C03594=1032.274,-117.414,-80.642,167.484,40.656,157.552
C03595=1032.267,-117.664,-80.633,167.481,40.657,157.552
C03596=1032.262,-117.914,-80.624,167.478,40.658,157.552
C03597=1032.256,-118.163,-80.615,167.476,40.660,157.553
C03598=1032.250,-118.414,-80.606,167.473,40.662,157.553
C03599=1032.245,-118.663,-80.597,167.470,40.663,157.553
C03600=1032.238,-118.913,-80.589,167.467,40.665,157.553
C03601=1032.232,-119.163,-80.579,167.465,40.667,157.553
C03602=1032.226,-119.412,-80.571,167.461,40.668,157.553
C03603=1032.220,-119.662,-80.561,167.458,40.669,157.553
C03604=1032.215,-119.912,-80.553,167.455,40.671,157.553
C03605=1032.208,-120.162,-80.544,167.452,40.673,157.554
C03606=1032.203,-120.411,-80.535,167.450,40.674,157.554
C03607=1032.197,-120.662,-80.526,167.447,40.676,157.554
C03608=1032.191,-120.911,-80.517,167.444,40.678,157.554
C03609=1032.186,-121.161,-80.508,167.441,40.679,157.554
C03610=1032.179,-121.411,-80.499,167.439,40.681,157.554
C03611=1032.173,-121.660,-80.491,167.436,40.682,157.554
C03612=1032.168,-121.911,-80.482,167.433,40.684,157.555
C03613=1032.162,-122.160,-80.473,167.430,40.685,157.555
C03614=1032.155,-122.410,-80.464,167.428,40.687,157.555
C03615=1032.150,-122.660,-80.456,167.425,40.689,157.555
C03616=1032.144,-122.909,-80.446,167.422,40.690,157.555
C03617=1032.139,-123.159,-80.438,167.419,40.692,157.555
C03618=1032.132,-123.409,-80.430,167.417,40.694,157.555
C03619=1032.126,-123.658,-80.420,167.414,40.695,157.556
C03620=1032.121,-123.909,-80.412,167.410,40.697,157.556
C03621=1032.115,-124.158,-80.403,167.407,40.699,157.556
C03622=1032.109,-124.407,-80.394,167.405,40.701,157.556
C03623=1032.103,-124.658,-80.386,167.402,40.702,157.556
C03624=1032.098,-124.907,-80.377,167.399,40.704,157.556
C03625=1032.091,-125.158,-80.369,167.396,40.706,157.556
C03626=1032.086,-125.407,-80.360,167.394,40.707,157.557
C03627=1032.079,-125.657,-80.351,167.391,40.709,157.557
C03628=1032.074,-125.906,-80.343,167.388,40.711,157.557
C03629=1032.068,-126.157,-80.334,167.385,40.712,157.557
C03630=1032.062,-126.406,-80.326,167.383,40.714,157.557
C03631=1032.056,-126.656,-80.317,167.380,40.716,157.557
C03632=1032.051,-126.906,-80.308,167.376,40.717,157.558
C03633=1032.045,-127.155,-80.300,167.373,40.719,157.558
C03634=1032.039,-127.406,-80.291,167.371,40.721,157.558
C03635=1032.033,-127.655,-80.283,167.368,40.722,157.558
C03636=1032.027,-127.904,-80.274,167.365,40.724,157.558
C03637=1032.022,-128.154,-80.266,167.362,40.725,157.558
C03638=1032.017,-128.403,-80.256,167.360,40.726,157.558
C03639=1032.014,-128.653,-80.245,167.357,40.726,157.558
C03640=1032.010,-128.903,-80.235,167.355,40.727,157.558
C03641=1032.008,-129.153,-80.223,167.353,40.725,157.558
C03642=1032.006,-129.403,-80.211,167.351,40.724,157.557
C03643=1032.004,-129.653,-80.199,167.348,40.723,157.557
C03644=1032.004,-129.903,-80.185,167.346,40.721,157.557
C03645=1032.004,-130.152,-80.171,167.344,40.719,157.556
C03646=1032.005,-130.402,-80.157,167.343,40.715,157.556
C03647=1032.006,-130.653,-80.142,167.341,40.712,157.555
C03648=1032.008,-130.902,-80.127,167.339,40.709,157.554
C03649=1032.011,-131.152,-80.111,167.337,40.704,157.553
C03650=1032.014,-131.402,-80.094,167.336,40.699,157.553
C03651=1032.018,-131.653,-80.077,167.335,40.694,157.552
C03652=1032.023,-131.902,-80.059,167.334,40.688,157.551
C03653=1032.029,-132.152,-80.041,167.332,40.682,157.550
C03654=1031.703,-132.177,-80.335,167.284,40.914,157.586
C03655=1031.699,-131.927,-80.354,167.284,40.920,157.587
C03656=1031.694,-131.678,-80.372,167.285,40.927,157.588
C03657=1031.690,-131.428,-80.389,167.288,40.932,157.589
C03658=1031.686,-131.177,-80.406,167.289,40.937,157.590
C03659=1031.683,-130.928,-80.422,167.291,40.941,157.591
C03660=1031.681,-130.677,-80.437,167.291,40.945,157.591
C03661=1031.680,-130.428,-80.452,167.293,40.948,157.592
C03662=1031.679,-130.177,-80.467,167.295,40.951,157.593
C03663=1031.679,-129.927,-80.480,167.298,40.953,157.593
C03664=1031.680,-129.678,-80.494,167.299,40.955,157.594
C03665=1031.681,-129.428,-80.506,167.301,40.957,157.594
C03666=1031.683,-129.178,-80.518,167.304,40.958,157.594
C03667=1031.685,-128.928,-80.529,167.306,40.959,157.594
C03668=1031.689,-128.678,-80.540,167.309,40.959,157.595
C03669=1031.693,-128.428,-80.551,167.311,40.959,157.595
C03670=1031.696,-128.179,-80.561,167.314,40.958,157.595
C03671=1031.702,-127.929,-80.570,167.317,40.956,157.595
C03672=1031.708,-127.679,-80.578,167.320,40.954,157.594
C03673=1031.714,-127.430,-80.587,167.322,40.953,157.594
C03674=1031.719,-127.181,-80.595,167.325,40.951,157.594
C03675=1031.726,-126.931,-80.604,167.328,40.949,157.594
C03676=1031.731,-126.681,-80.612,167.331,40.948,157.594
C03677=1031.736,-126.431,-80.621,167.333,40.946,157.594
C03678=1031.743,-126.182,-80.629,167.336,40.944,157.594
C03679=1031.748,-125.932,-80.638,167.339,40.942,157.593
C03680=1031.755,-125.682,-80.646,167.343,40.941,157.593
C03681=1031.760,-125.432,-80.655,167.345,40.939,157.593
C03682=1031.766,-125.182,-80.664,167.348,40.937,157.593
C03683=1031.772,-124.933,-80.672,167.351,40.936,157.593
C03684=1031.778,-124.683,-80.681,167.353,40.934,157.593
C03685=1031.784,-124.433,-80.690,167.356,40.932,157.593
C03686=1031.790,-124.183,-80.697,167.359,40.931,157.592
C03687=1031.796,-123.934,-80.707,167.362,40.929,157.592
C03688=1031.801,-123.684,-80.715,167.364,40.927,157.592
C03689=1031.807,-123.434,-80.724,167.367,40.925,157.592
C03690=1031.813,-123.184,-80.732,167.371,40.924,157.592
C03691=1031.819,-122.934,-80.742,167.374,40.922,157.592
C03692=1031.824,-122.685,-80.750,167.376,40.920,157.592
C03693=1031.831,-122.434,-80.759,167.379,40.919,157.591
C03694=1031.837,-122.185,-80.768,167.382,40.917,157.591
C03695=1031.842,-121.935,-80.777,167.385,40.915,157.591
C03696=1031.848,-121.686,-80.786,167.387,40.913,157.591
C03697=1031.854,-121.435,-80.795,167.390,40.912,157.591
C03698=1031.860,-121.186,-80.803,167.393,40.910,157.591
C03699=1031.866,-120.936,-80.812,167.396,40.908,157.591
C03700=1031.871,-120.687,-80.821,167.398,40.907,157.590
C03701=1031.877,-120.436,-80.829,167.401,40.905,157.590
C03702=1031.883,-120.187,-80.838,167.405,40.903,157.590
C03703=1031.888,-119.973,-80.846,167.407,40.902,157.590
C03704=1031.893,-119.760,-80.854,167.409,40.901,157.590
C03705=1031.898,-119.546,-80.861,167.411,40.899,157.590
C03706=1031.903,-119.332,-80.869,167.414,40.898,157.590
C03707=1031.908,-119.118,-80.876,167.417,40.896,157.590
C03708=1031.914,-118.904,-80.884,167.419,40.895,157.589
C03709=1031.918,-118.690,-80.892,167.421,40.894,157.589
C03710=1031.924,-118.477,-80.899,167.424,40.892,157.589
C03711=1031.929,-118.226,-80.908,167.427,40.890,157.589
C03712=1031.936,-117.977,-80.918,167.430,40.889,157.589
C03713=1031.942,-117.727,-80.926,167.432,40.887,157.589
C03714=1031.948,-117.477,-80.935,167.435,40.885,157.589
C03715=1031.956,-117.119,-80.949,167.439,40.884,157.589
C03716=1031.965,-116.761,-80.961,167.443,40.881,157.588
C03717=1031.973,-116.403,-80.974,167.447,40.878,157.588
C03718=1031.981,-116.044,-80.987,167.452,40.877,157.588
C03719=1031.987,-115.794,-80.996,167.455,40.875,157.588
C03720=1031.994,-115.544,-81.005,167.457,40.873,157.588
C03721=1031.999,-115.295,-81.014,167.460,40.872,157.588
C03722=1032.005,-115.045,-81.023,167.463,40.870,157.587
C03723=1032.011,-114.795,-81.033,167.466,40.868,157.587
C03724=1032.016,-114.545,-81.041,167.468,40.867,157.587
C03725=1032.023,-114.295,-81.051,167.471,40.865,157.587
C03726=1032.029,-114.045,-81.060,167.474,40.864,157.587
C03727=1032.034,-113.796,-81.069,167.477,40.862,157.587
C03728=1032.040,-113.546,-81.078,167.479,40.860,157.587
C03729=1032.046,-113.296,-81.087,167.482,40.859,157.587
C03730=1032.052,-113.047,-81.096,167.485,40.858,157.586
C03731=1032.058,-112.797,-81.106,167.488,40.856,157.586
C03732=1032.064,-112.547,-81.116,167.491,40.854,157.586
C03733=1032.069,-112.297,-81.124,167.493,40.853,157.586
C03734=1032.075,-112.047,-81.134,167.496,40.852,157.586
C03735=1032.082,-111.798,-81.143,167.499,40.850,157.586
C03736=1032.087,-111.549,-81.152,167.502,40.848,157.586
C03737=1032.093,-111.298,-81.161,167.504,40.847,157.586
C03738=1032.099,-111.048,-81.171,167.508,40.846,157.586
C03739=1032.105,-110.799,-81.180,167.511,40.844,157.585
C03740=1032.111,-110.549,-81.190,167.514,40.842,157.585
C03741=1032.117,-110.299,-81.198,167.516,40.840,157.585
C03742=1032.123,-110.049,-81.208,167.519,40.839,157.585
C03743=1032.129,-109.799,-81.218,167.522,40.838,157.585
C03744=1032.135,-109.550,-81.227,167.525,40.836,157.585
C03745=1032.141,-109.301,-81.236,167.528,40.834,157.585
C03746=1032.147,-109.051,-81.246,167.530,40.833,157.585
C03747=1032.153,-108.800,-81.255,167.533,40.832,157.584
C03748=1032.159,-108.551,-81.264,167.536,40.830,157.584
C03749=1032.165,-108.301,-81.274,167.539,40.828,157.584
C03750=1032.171,-108.052,-81.283,167.542,40.827,157.584
C03751=1032.177,-107.802,-81.293,167.544,40.826,157.584
C03752=1032.183,-107.552,-81.302,167.547,40.824,157.584
C03753=1032.189,-107.302,-81.312,167.550,40.822,157.584
C03754=1032.195,-107.053,-81.321,167.553,40.821,157.584
C03755=1032.200,-106.803,-81.331,167.555,40.820,157.583
C03756=1032.206,-106.553,-81.340,167.558,40.818,157.583
C03757=1032.212,-106.303,-81.350,167.561,40.817,157.583
C03758=1032.219,-106.053,-81.359,167.564,40.815,157.583
C03759=1032.224,-105.804,-81.368,167.567,40.814,157.583
C03760=1032.230,-105.554,-81.378,167.569,40.813,157.583
C03761=1032.236,-105.304,-81.388,167.572,40.811,157.583
C03762=1032.242,-105.054,-81.398,167.575,40.810,157.583
C03763=1032.248,-104.804,-81.407,167.578,40.808,157.583
C03764=1032.254,-104.555,-81.417,167.581,40.807,157.582
C03765=1032.260,-104.306,-81.426,167.583,40.806,157.582
C03766=1032.265,-104.055,-81.436,167.586,40.804,157.582
C03767=1032.272,-103.806,-81.446,167.589,40.803,157.582
C03768=1032.278,-103.556,-81.456,167.592,40.801,157.582
C03769=1032.284,-103.307,-81.466,167.595,40.800,157.582
C03770=1032.290,-103.057,-81.475,167.597,40.799,157.582
C03771=1032.296,-102.807,-81.485,167.600,40.797,157.582
C03772=1032.302,-102.557,-81.495,167.603,40.796,157.582
C03773=1032.308,-102.307,-81.504,167.606,40.794,157.582
C03774=1032.314,-102.058,-81.514,167.609,40.793,157.581
C03775=1032.319,-101.808,-81.524,167.611,40.792,157.581
C03776=1032.325,-101.558,-81.533,167.614,40.790,157.581
C03777=1032.332,-101.309,-81.544,167.617,40.789,157.581
C03778=1032.338,-101.059,-81.553,167.620,40.787,157.581
C03779=1032.344,-100.772,-81.565,167.624,40.785,157.581
C03780=1032.351,-100.485,-81.576,167.626,40.784,157.581
C03781=1032.358,-100.198,-81.587,167.629,40.783,157.581
C03782=1032.365,-99.911,-81.598,167.633,40.781,157.581
C03783=1032.371,-99.661,-81.608,167.636,40.779,157.580
C03784=1032.377,-99.412,-81.618,167.639,40.778,157.580
C03785=1032.383,-99.162,-81.628,167.641,40.777,157.580
C03786=1032.389,-98.912,-81.638,167.644,40.775,157.580
C03787=1032.395,-98.662,-81.648,167.647,40.774,157.580
C03788=1032.401,-98.413,-81.658,167.650,40.772,157.580
C03789=1032.408,-98.163,-81.668,167.653,40.771,157.580
C03790=1032.414,-97.913,-81.677,167.655,40.770,157.580
C03791=1032.419,-97.663,-81.687,167.658,40.768,157.580
C03792=1032.426,-97.414,-81.698,167.661,40.767,157.580
C03793=1032.431,-97.164,-81.708,167.664,40.766,157.580
C03794=1032.437,-96.914,-81.717,167.667,40.764,157.579
C03795=1032.443,-96.665,-81.728,167.670,40.763,157.579
C03796=1032.449,-96.415,-81.738,167.672,40.762,157.579
C03797=1032.455,-96.165,-81.748,167.674,40.761,157.579
C03798=1032.461,-95.916,-81.758,167.677,40.760,157.579
C03799=1032.466,-95.665,-81.768,167.680,40.758,157.579
C03800=1032.473,-95.416,-81.779,167.683,40.757,157.579
C03801=1032.478,-95.166,-81.789,167.686,40.756,157.579
C03802=1032.485,-94.916,-81.798,167.688,40.754,157.579
C03803=1032.490,-94.667,-81.809,167.691,40.753,157.579
C03804=1032.496,-94.417,-81.819,167.694,40.752,157.579
C03805=1032.502,-94.168,-81.830,167.697,40.751,157.579
C03806=1032.508,-93.918,-81.839,167.700,40.750,157.579
C03807=1032.514,-93.668,-81.850,167.702,40.748,157.578
C03808=1032.520,-93.417,-81.861,167.705,40.747,157.578
C03809=1032.527,-93.168,-81.871,167.708,40.746,157.578
C03810=1032.532,-92.918,-81.881,167.711,40.744,157.578
C03811=1032.539,-92.669,-81.891,167.714,40.743,157.578
C03812=1032.544,-92.419,-81.902,167.716,40.742,157.578
C03813=1032.550,-92.170,-81.912,167.718,40.741,157.578
C03814=1032.556,-91.920,-81.922,167.721,40.740,157.578
C03815=1032.562,-91.670,-81.932,167.724,40.738,157.578
C03816=1032.568,-91.420,-81.942,167.727,40.737,157.578
C03817=1032.574,-91.171,-81.953,167.730,40.736,157.578
C03818=1032.580,-90.921,-81.963,167.733,40.734,157.577
C03819=1032.586,-90.671,-81.974,167.736,40.733,157.577
C03820=1032.593,-90.422,-81.984,167.738,40.732,157.577
C03821=1032.598,-90.172,-81.995,167.741,40.731,157.577
C03822=1032.604,-89.922,-82.005,167.744,40.730,157.577
C03823=1032.610,-89.672,-82.015,167.747,40.728,157.577
C03824=1032.616,-89.423,-82.025,167.750,40.727,157.577
C03825=1032.622,-89.174,-82.036,167.752,40.726,157.577
C03826=1032.628,-88.923,-82.047,167.754,40.725,157.577
C03827=1032.635,-88.674,-82.057,167.757,40.724,157.577
C03828=1032.640,-88.423,-82.067,167.760,40.723,157.577
C03829=1032.647,-88.174,-82.077,167.763,40.721,157.577
C03830=1032.652,-87.925,-82.088,167.766,40.720,157.577
C03831=1032.658,-87.674,-82.099,167.768,40.718,157.576
C03832=1032.665,-87.425,-82.109,167.771,40.717,157.576
C03833=1032.671,-87.175,-82.120,167.774,40.716,157.576
C03834=1032.677,-86.926,-82.130,167.777,40.715,157.576
C03835=1032.682,-86.676,-82.140,167.780,40.714,157.576
C03836=1032.689,-86.426,-82.151,167.783,40.713,157.576
C03837=1032.695,-86.177,-82.162,167.786,40.711,157.576
C03838=1032.701,-85.927,-82.172,167.787,40.710,157.576
C03839=1032.707,-85.677,-82.182,167.790,40.709,157.576
C03840=1032.713,-85.427,-82.194,167.793,40.707,157.576
C03841=1032.720,-85.178,-82.204,167.796,40.706,157.576
C03842=1032.725,-84.928,-82.214,167.799,40.705,157.576
C03843=1032.732,-84.643,-82.226,167.802,40.704,157.576
C03844=1032.740,-84.359,-82.239,167.805,40.703,157.575
C03845=1032.746,-84.074,-82.251,167.808,40.701,157.575
C03846=1032.753,-83.789,-82.263,167.811,40.699,157.575
C03847=1032.760,-83.539,-82.274,167.814,40.698,157.575
C03848=1032.766,-83.289,-82.284,167.817,40.697,157.575
C03849=1032.771,-83.040,-82.295,167.819,40.696,157.575
C03850=1032.779,-82.790,-82.305,167.822,40.695,157.575
C03851=1032.784,-82.540,-82.316,167.825,40.694,157.575
C03852=1032.790,-82.291,-82.327,167.828,40.692,157.575
C03853=1032.797,-82.041,-82.338,167.831,40.691,157.575
C03854=1032.803,-81.792,-82.349,167.834,40.690,157.575
C03855=1032.809,-81.542,-82.358,167.837,40.688,157.575
C03856=1032.815,-81.292,-82.369,167.839,40.687,157.574
C03857=1032.821,-81.042,-82.380,167.841,40.687,157.574
C03858=1032.828,-80.793,-82.391,167.844,40.685,157.574
C03859=1032.834,-80.543,-82.402,167.847,40.684,157.574
C03860=1032.840,-80.293,-82.413,167.850,40.683,157.574
C03861=1032.846,-80.044,-82.423,167.853,40.681,157.574
C03862=1032.852,-79.794,-82.434,167.855,40.680,157.574
C03863=1032.858,-79.544,-82.445,167.858,40.679,157.574
C03864=1032.864,-79.295,-82.456,167.861,40.678,157.574
C03865=1032.870,-79.045,-82.467,167.863,40.677,157.574
C03866=1032.876,-78.795,-82.478,167.866,40.676,157.574
C03867=1032.883,-78.545,-82.489,167.869,40.675,157.574
C03868=1032.889,-78.296,-82.500,167.872,40.674,157.574
C03869=1032.895,-78.046,-82.510,167.875,40.673,157.574
C03870=1032.901,-77.796,-82.522,167.877,40.672,157.574
C03871=1032.907,-77.547,-82.533,167.880,40.671,157.574
C03872=1032.912,-77.297,-82.543,167.882,40.670,157.573
C03873=1032.919,-77.047,-82.555,167.885,40.668,157.573
C03874=1032.924,-76.797,-82.566,167.888,40.667,157.573
C03875=1032.932,-76.548,-82.577,167.891,40.666,157.573
C03876=1032.938,-76.299,-82.588,167.894,40.665,157.573
///RCONF 1,0,0,1,0,0,0,0,0,0,0,0,0,0,0,0,0,0,0,0,0,0,0,0
C03877=1032.943,-76.049,-82.599,167.896,40.664,157.573
C03878=1032.950,-75.799,-82.610,167.899,40.663,157.573
C03879=1032.955,-75.550,-82.621,167.901,40.662,157.573
C03880=1032.962,-75.299,-82.632,167.904,40.661,157.573
C03881=1032.968,-75.050,-82.643,167.907,40.660,157.573
C03882=1032.974,-74.800,-82.655,167.910,40.659,157.573
C03883=1032.980,-74.551,-82.666,167.913,40.658,157.573
C03884=1032.986,-74.301,-82.677,167.916,40.657,157.573
C03885=1032.992,-74.051,-82.688,167.917,40.656,157.573
C03886=1032.998,-73.801,-82.699,167.920,40.655,157.573
C03887=1033.004,-73.552,-82.711,167.923,40.654,157.573
C03888=1033.010,-73.303,-82.722,167.926,40.653,157.573
C03889=1033.016,-73.052,-82.733,167.929,40.652,157.573
C03890=1033.022,-72.803,-82.744,167.931,40.651,157.573
C03891=1033.028,-72.553,-82.756,167.934,40.650,157.572
C03892=1033.034,-72.303,-82.767,167.937,40.649,157.572
C03893=1033.040,-72.054,-82.779,167.940,40.648,157.572
C03894=1033.046,-71.804,-82.790,167.941,40.647,157.572
C03895=1033.053,-71.554,-82.801,167.944,40.646,157.572
C03896=1033.058,-71.305,-82.813,167.947,40.645,157.572
C03897=1033.064,-71.055,-82.825,167.950,40.644,157.572
///RCONF 1,0,0,0,0,0,0,0,0,0,0,0,0,0,0,0,0,0,0,0,0,0,0,0
C03898=1033.070,-70.805,-82.836,167.953,40.643,157.572
C03899=1033.077,-70.556,-82.848,167.955,40.642,157.572
C03900=1033.082,-70.306,-82.858,167.958,40.642,157.572
C03901=1033.088,-70.056,-82.871,167.961,40.641,157.572
C03902=1033.094,-69.807,-82.882,167.964,40.640,157.572
C03903=1033.100,-69.557,-82.893,167.966,40.639,157.572
C03904=1033.106,-69.308,-82.905,167.968,40.638,157.572
C03905=1033.113,-69.058,-82.916,167.971,40.637,157.572
C03906=1033.118,-68.808,-82.928,167.974,40.636,157.572
C03907=1033.125,-68.526,-82.941,167.977,40.635,157.572
C03908=1033.132,-68.243,-82.954,167.980,40.634,157.572
C03909=1033.139,-67.961,-82.967,167.983,40.633,157.572
C03910=1033.146,-67.677,-82.980,167.986,40.632,157.572
C03911=1033.151,-67.428,-82.991,167.989,40.631,157.572
C03912=1033.158,-67.178,-83.003,167.992,40.630,157.572
C03913=1033.164,-66.929,-83.014,167.994,40.629,157.572
C03914=1033.170,-66.679,-83.026,167.996,40.629,157.572
C03915=1033.176,-66.429,-83.037,167.999,40.628,157.572
C03916=1033.182,-66.180,-83.050,168.002,40.627,157.572
C03917=1033.189,-65.930,-83.062,168.005,40.626,157.572
C03918=1033.194,-65.681,-83.072,168.007,40.625,157.571
C03919=1033.201,-65.431,-83.084,168.010,40.624,157.571
C03920=1033.206,-65.181,-83.096,168.013,40.623,157.571
C03921=1033.213,-64.932,-83.108,168.016,40.622,157.571
C03922=1033.219,-64.681,-83.119,168.017,40.621,157.571
C03923=1033.225,-64.433,-83.131,168.020,40.620,157.571
C03924=1033.231,-64.183,-83.143,168.023,40.619,157.571
C03925=1033.237,-63.932,-83.154,168.026,40.618,157.571
C03926=1033.243,-63.684,-83.166,168.028,40.617,157.571
C03927=1033.250,-63.433,-83.177,168.031,40.616,157.571
C03928=1033.256,-63.184,-83.189,168.034,40.615,157.571
C03929=1033.262,-62.935,-83.201,168.037,40.615,157.571
C03930=1033.268,-62.684,-83.213,168.040,40.614,157.571
C03931=1033.275,-62.435,-83.225,168.042,40.613,157.571
C03932=1033.281,-62.186,-83.236,168.044,40.612,157.571
C03933=1033.286,-61.935,-83.248,168.047,40.611,157.571
C03934=1033.293,-61.686,-83.260,168.050,40.610,157.571
C03935=1033.299,-61.437,-83.272,168.052,40.609,157.571
C03936=1033.305,-61.187,-83.283,168.055,40.608,157.571
C03937=1033.311,-60.937,-83.295,168.058,40.607,157.571
C03938=1033.318,-60.687,-83.307,168.061,40.606,157.571
C03939=1033.324,-60.438,-83.318,168.063,40.605,157.571
C03940=1033.330,-60.188,-83.331,168.066,40.604,157.571
C03941=1033.336,-59.938,-83.343,168.068,40.603,157.571
C03942=1033.343,-59.689,-83.355,168.071,40.602,157.571
C03943=1033.349,-59.439,-83.366,168.073,40.602,157.570
C03944=1033.354,-59.190,-83.378,168.076,40.601,157.570
C03945=1033.361,-58.940,-83.390,168.079,40.600,157.570
C03946=1033.368,-58.690,-83.402,168.082,40.599,157.571
C03947=1033.373,-58.441,-83.414,168.084,40.598,157.570
C03948=1033.379,-58.191,-83.425,168.087,40.597,157.570
C03949=1033.386,-57.941,-83.437,168.090,40.596,157.570
C03950=1033.393,-57.692,-83.449,168.092,40.596,157.570
C03951=1033.399,-57.442,-83.462,168.094,40.595,157.570
C03952=1033.405,-57.193,-83.474,168.097,40.594,157.570
C03953=1033.411,-56.943,-83.485,168.100,40.593,157.570
C03954=1033.417,-56.693,-83.497,168.102,40.592,157.570
C03955=1033.424,-56.443,-83.509,168.105,40.591,157.570
C03956=1033.430,-56.194,-83.521,168.108,40.590,157.570
C03957=1033.436,-55.945,-83.533,168.111,40.589,157.570
C03958=1033.442,-55.695,-83.545,168.113,40.588,157.570
C03959=1033.449,-55.446,-83.557,168.116,40.587,157.570
C03960=1033.455,-55.195,-83.569,168.118,40.586,157.570
C03961=1033.461,-54.945,-83.581,168.121,40.585,157.570
C03962=1033.468,-54.696,-83.593,168.123,40.585,157.570
C03963=1033.474,-54.446,-83.605,168.126,40.584,157.570
C03964=1033.480,-54.197,-83.617,168.129,40.583,157.570
C03965=1033.486,-53.948,-83.629,168.132,40.582,157.570
C03966=1033.493,-53.698,-83.641,168.134,40.581,157.570
C03967=1033.499,-53.448,-83.654,168.137,40.580,157.570
C03968=1033.505,-53.199,-83.666,168.140,40.579,157.570
C03969=1033.512,-52.949,-83.678,168.142,40.578,157.570
C03970=1033.519,-52.699,-83.690,168.144,40.577,157.570
C03971=1033.525,-52.418,-83.703,168.147,40.576,157.569
C03972=1033.533,-52.137,-83.717,168.150,40.575,157.569
C03973=1033.540,-51.855,-83.731,168.153,40.574,157.569
C03974=1033.547,-51.574,-83.744,168.156,40.573,157.569
C03975=1033.553,-51.324,-83.757,168.159,40.572,157.569
C03976=1033.560,-51.075,-83.769,168.162,40.571,157.569
C03977=1033.566,-50.825,-83.781,168.165,40.570,157.569
C03978=1033.572,-50.575,-83.794,168.167,40.569,157.569
C03979=1033.579,-50.326,-83.806,168.169,40.568,157.569
C03980=1033.585,-50.076,-83.818,168.173,40.568,157.569
C03981=1033.591,-49.826,-83.831,168.174,40.567,157.569
C03982=1033.597,-49.576,-83.843,168.177,40.566,157.569
C03983=1033.603,-49.327,-83.855,168.180,40.566,157.569
C03984=1033.609,-49.078,-83.868,168.182,40.565,157.569
C03985=1033.616,-48.828,-83.880,168.185,40.564,157.569
C03986=1033.621,-48.578,-83.893,168.187,40.563,157.569
C03987=1033.627,-48.329,-83.905,168.190,40.563,157.569
C03988=1033.634,-48.079,-83.917,168.193,40.562,157.569
C03989=1033.640,-47.830,-83.930,168.195,40.561,157.569
C03990=1033.646,-47.580,-83.943,168.198,40.561,157.569
C03991=1033.652,-47.330,-83.955,168.201,40.560,157.569
C03992=1033.659,-47.080,-83.967,168.203,40.559,157.569
C03993=1033.665,-46.831,-83.981,168.206,40.559,157.569
C03994=1033.671,-46.581,-83.993,168.209,40.558,157.569
C03995=1033.677,-46.332,-84.005,168.210,40.557,157.569
C03996=1033.683,-46.082,-84.018,168.213,40.556,157.569
C03997=1033.690,-45.833,-84.031,168.215,40.556,157.569
C03998=1033.696,-45.583,-84.043,168.218,40.555,157.569
C03999=1033.702,-45.333,-84.056,168.221,40.554,157.569
C04000=1033.708,-45.084,-84.069,168.223,40.553,157.569
C04001=1033.714,-44.834,-84.081,168.226,40.552,157.569
C04002=1033.721,-44.584,-84.093,168.229,40.551,157.569
C04003=1033.727,-44.335,-84.107,168.231,40.551,157.569
C04004=1033.733,-44.085,-84.119,168.234,40.550,157.569
C04005=1033.740,-43.836,-84.131,168.236,40.549,157.569
C04006=1033.746,-43.586,-84.144,168.239,40.549,157.569
C04007=1033.752,-43.337,-84.157,168.242,40.548,157.569
C04008=1033.758,-43.087,-84.170,168.244,40.547,157.569
C04009=1033.765,-42.838,-84.182,168.246,40.546,157.569
C04010=1033.771,-42.588,-84.195,168.249,40.546,157.569
C04011=1033.777,-42.339,-84.208,168.251,40.545,157.569
C04012=1033.783,-42.089,-84.221,168.254,40.544,157.569
C04013=1033.790,-41.840,-84.233,168.256,40.544,157.569
C04014=1033.796,-41.590,-84.246,168.259,40.543,157.569
C04015=1033.802,-41.339,-84.259,168.262,40.542,157.569
C04016=1033.808,-41.090,-84.272,168.264,40.542,157.569
C04017=1033.815,-40.840,-84.284,168.267,40.541,157.569
C04018=1033.821,-40.591,-84.297,168.270,40.540,157.569
C04019=1033.827,-40.341,-84.310,168.272,40.539,157.569
C04020=1033.833,-40.092,-84.323,168.275,40.539,157.569
C04021=1033.840,-39.842,-84.335,168.277,40.538,157.569
C04022=1033.846,-39.593,-84.348,168.279,40.537,157.569
C04023=1033.852,-39.343,-84.361,168.283,40.536,157.569
C04024=1033.859,-39.093,-84.374,168.284,40.536,157.569
C04025=1033.865,-38.844,-84.386,168.287,40.535,157.569
C04026=1033.872,-38.594,-84.400,168.289,40.534,157.569
C04027=1033.878,-38.345,-84.412,168.292,40.533,157.569
C04028=1033.884,-38.095,-84.426,168.295,40.533,157.569
C04029=1033.890,-37.846,-84.439,168.297,40.532,157.569
C04030=1033.896,-37.596,-84.451,168.300,40.531,157.569
C04031=1033.903,-37.346,-84.465,168.302,40.531,157.569
C04032=1033.909,-37.097,-84.478,168.305,40.530,157.569
C04033=1033.915,-36.847,-84.491,168.307,40.530,157.569
C04034=1033.921,-36.598,-84.504,168.310,40.529,157.569
C04035=1033.928,-36.316,-84.519,168.313,40.529,157.569
C04036=1033.935,-36.036,-84.534,168.316,40.528,157.569
C04037=1033.942,-35.755,-84.548,168.319,40.527,157.569
C04038=1033.948,-35.474,-84.563,168.321,40.526,157.569
C04039=1033.954,-35.224,-84.576,168.324,40.526,157.569
C04040=1033.961,-34.974,-84.590,168.327,40.525,157.569
C04041=1033.967,-34.724,-84.602,168.328,40.524,157.569
C04042=1033.973,-34.475,-84.616,168.332,40.524,157.569
C04043=1033.979,-34.226,-84.629,168.333,40.523,157.569
C04044=1033.986,-33.977,-84.642,168.336,40.522,157.569
C04045=1033.992,-33.726,-84.655,168.338,40.522,157.569
C04046=1033.998,-33.477,-84.668,168.341,40.521,157.569
C04047=1034.005,-33.228,-84.682,168.343,40.521,157.569
C04048=1034.011,-32.978,-84.695,168.346,40.520,157.569
C04049=1034.017,-32.728,-84.708,168.348,40.520,157.569
C04050=1034.024,-32.478,-84.721,168.351,40.519,157.569
C04051=1034.030,-32.229,-84.734,168.354,40.518,157.569
C04052=1034.036,-31.980,-84.748,168.356,40.517,157.569
C04053=1034.043,-31.730,-84.761,168.359,40.516,157.569
C04054=1034.049,-31.480,-84.774,168.361,40.516,157.569
C04055=1034.055,-31.231,-84.787,168.364,40.515,157.569
C04056=1034.061,-30.982,-84.800,168.366,40.515,157.569
C04057=1034.068,-30.732,-84.814,168.369,40.514,157.569
C04058=1034.074,-30.482,-84.827,168.371,40.514,157.569
C04059=1034.080,-30.233,-84.841,168.374,40.513,157.569
C04060=1034.087,-29.984,-84.854,168.375,40.512,157.569
C04061=1034.093,-29.733,-84.867,168.379,40.512,157.569
C04062=1034.099,-29.484,-84.880,168.380,40.511,157.569
C04063=1034.106,-29.235,-84.893,168.383,40.511,157.569
C04064=1034.112,-28.985,-84.907,168.386,40.510,157.569
C04065=1034.119,-28.735,-84.920,168.388,40.509,157.569
C04066=1034.125,-28.486,-84.933,168.391,40.508,157.569
C04067=1034.131,-28.236,-84.948,168.393,40.508,157.569
C04068=1034.137,-27.987,-84.961,168.396,40.507,157.569
C04069=1034.143,-27.737,-84.974,168.398,40.506,157.569
C04070=1034.150,-27.487,-84.988,168.401,40.506,157.569
C04071=1034.156,-27.238,-85.001,168.403,40.505,157.569
C04072=1034.163,-26.989,-85.014,168.406,40.505,157.569
C04073=1034.169,-26.739,-85.028,168.408,40.504,157.569
C04074=1034.175,-26.489,-85.042,168.411,40.504,157.569
C04075=1034.181,-26.240,-85.055,168.413,40.503,157.569
C04076=1034.188,-25.990,-85.069,168.416,40.503,157.569
C04077=1034.193,-25.741,-85.083,168.418,40.502,157.569
C04078=1034.200,-25.491,-85.096,168.421,40.501,157.569
C04079=1034.206,-25.241,-85.110,168.423,40.501,157.569
C04080=1034.213,-24.992,-85.123,168.426,40.500,157.569
C04081=1034.218,-24.742,-85.137,168.428,40.500,157.569
C04082=1034.225,-24.492,-85.150,168.431,40.499,157.569
C04083=1034.231,-24.243,-85.164,168.433,40.499,157.569
C04084=1034.237,-23.993,-85.178,168.435,40.499,157.569
C04085=1034.243,-23.744,-85.191,168.437,40.498,157.569
C04086=1034.250,-23.495,-85.205,168.440,40.497,157.569
C04087=1034.256,-23.245,-85.219,168.442,40.497,157.569
C04088=1034.262,-22.995,-85.233,168.444,40.496,157.569
C04089=1034.268,-22.746,-85.246,168.447,40.496,157.569
C04090=1034.274,-22.496,-85.260,168.449,40.495,157.569
C04091=1034.281,-22.247,-85.273,168.452,40.495,157.569
C04092=1034.288,-21.997,-85.288,168.454,40.494,157.569
C04093=1034.293,-21.748,-85.302,168.457,40.494,157.569
C04094=1034.300,-21.499,-85.315,168.459,40.493,157.569
C04095=1034.306,-21.249,-85.329,168.462,40.492,157.569
C04096=1034.312,-20.999,-85.342,168.464,40.492,157.569
C04097=1034.319,-20.750,-85.357,168.467,40.491,157.569
C04098=1034.325,-20.500,-85.370,168.469,40.491,157.569
C04099=1034.332,-20.218,-85.385,168.472,40.490,157.569
C04100=1034.339,-19.937,-85.401,168.475,40.490,157.569
C04101=1034.347,-19.654,-85.417,168.477,40.489,157.569
C04102=1034.353,-19.373,-85.432,168.480,40.489,157.569
C04103=1034.360,-19.123,-85.446,168.483,40.488,157.569
C04104=1034.366,-18.874,-85.460,168.485,40.487,157.569
C04105=1034.373,-18.624,-85.474,168.487,40.487,157.569
C04106=1034.378,-18.375,-85.488,168.490,40.486,157.569
C04107=1034.385,-18.125,-85.502,168.492,40.485,157.569
C04108=1034.392,-17.876,-85.516,168.495,40.485,157.569
C04109=1034.398,-17.626,-85.530,168.497,40.485,157.569
C04110=1034.404,-17.377,-85.543,168.500,40.484,157.569
C04111=1034.411,-17.127,-85.557,168.502,40.484,157.569
C04112=1034.417,-16.878,-85.571,168.505,40.483,157.569
C04113=1034.423,-16.628,-85.585,168.507,40.483,157.569
C04114=1034.429,-16.379,-85.600,168.509,40.482,157.569
C04115=1034.436,-16.129,-85.613,168.511,40.481,157.569
C04116=1034.442,-15.880,-85.627,168.513,40.481,157.569
C04117=1034.449,-15.630,-85.641,168.516,40.480,157.569
C04118=1034.455,-15.380,-85.655,168.518,40.479,157.569
C04119=1034.461,-15.131,-85.670,168.521,40.479,157.569
C04120=1034.468,-14.881,-85.683,168.523,40.479,157.569
C04121=1034.474,-14.632,-85.698,168.525,40.479,157.569
C04122=1034.481,-14.382,-85.711,168.528,40.478,157.569
C04123=1034.486,-14.133,-85.726,168.530,40.477,157.569
C04124=1034.492,-13.883,-85.740,168.533,40.477,157.569
C04125=1034.499,-13.634,-85.754,168.535,40.476,157.569
C04126=1034.505,-13.384,-85.768,168.537,40.476,157.569
C04127=1034.511,-13.135,-85.783,168.540,40.476,157.569
C04128=1034.518,-12.885,-85.797,168.542,40.475,157.569
C04129=1034.523,-12.636,-85.811,168.545,40.475,157.570
C04130=1034.530,-12.386,-85.825,168.547,40.474,157.570
C04131=1034.537,-12.136,-85.840,168.549,40.474,157.569
C04132=1034.542,-11.887,-85.854,168.552,40.473,157.570
C04133=1034.549,-11.638,-85.868,168.554,40.473,157.570
C04134=1034.555,-11.389,-85.883,168.557,40.473,157.570
C04135=1034.562,-11.139,-85.896,168.559,40.472,157.570
C04136=1034.568,-10.890,-85.911,168.561,40.472,157.570
C04137=1034.574,-10.639,-85.925,168.564,40.471,157.570
C04138=1034.581,-10.390,-85.939,168.566,40.470,157.570
C04139=1034.587,-10.141,-85.954,168.569,40.470,157.570
C04140=1034.593,-9.891,-85.968,168.571,40.470,157.570
C04141=1034.600,-9.641,-85.983,168.573,40.469,157.570
C04142=1034.605,-9.392,-85.996,168.576,40.469,157.570
C04143=1034.612,-9.142,-86.011,168.578,40.469,157.570
C04144=1034.618,-8.894,-86.025,168.580,40.468,157.570
C04145=1034.624,-8.643,-86.040,168.583,40.467,157.570
C04146=1034.631,-8.394,-86.055,168.585,40.467,157.570
C04147=1034.637,-8.145,-86.069,168.588,40.466,157.570
C04148=1034.643,-7.895,-86.083,168.590,40.466,157.570
C04149=1034.650,-7.645,-86.097,168.592,40.466,157.570
C04150=1034.656,-7.396,-86.112,168.595,40.465,157.570
C04151=1034.662,-7.146,-86.126,168.597,40.465,157.570
C04152=1034.669,-6.897,-86.140,168.599,40.464,157.570
C04153=1034.675,-6.648,-86.155,168.602,40.464,157.570
C04154=1034.681,-6.398,-86.170,168.604,40.463,157.570
C04155=1034.688,-6.148,-86.183,168.607,40.463,157.570
C04156=1034.695,-5.899,-86.198,168.609,40.462,157.570
C04157=1034.700,-5.650,-86.213,168.611,40.462,157.570
C04158=1034.708,-5.400,-86.227,168.614,40.461,157.570
C04159=1034.714,-5.150,-86.242,168.616,40.461,157.570
C04160=1034.719,-4.901,-86.256,168.618,40.461,157.570
C04161=1034.727,-4.652,-86.271,168.620,40.460,157.570
C04162=1034.733,-4.402,-86.285,168.622,40.459,157.570
C04163=1034.740,-4.119,-86.302,168.626,40.459,157.570
C04164=1034.747,-3.835,-86.318,168.628,40.458,157.570
C04165=1034.754,-3.552,-86.335,168.630,40.458,157.570
C04166=1034.762,-3.269,-86.352,168.633,40.458,157.570
C04167=1034.768,-3.019,-86.367,168.635,40.457,157.570
C04168=1034.774,-2.769,-86.381,168.639,40.457,157.571
C04169=1034.780,-2.520,-86.395,168.640,40.456,157.570
C04170=1034.786,-2.270,-86.410,168.642,40.456,157.571
C04171=1034.793,-2.021,-86.425,168.644,40.456,157.571
C04172=1034.798,-1.772,-86.440,168.647,40.456,157.571
C04173=1034.805,-1.522,-86.455,168.650,40.455,157.571
C04174=1034.811,-1.272,-86.470,168.652,40.455,157.571
C04175=1034.817,-1.023,-86.485,168.654,40.454,157.571
C04176=1034.823,-0.774,-86.499,168.656,40.454,157.571
C04177=1034.830,-0.524,-86.514,168.658,40.454,157.571
C04178=1034.836,-0.274,-86.529,168.662,40.453,157.571
C04179=1034.842,-0.025,-86.544,168.664,40.453,157.571
C04180=1034.848,0.224,-86.559,168.666,40.453,157.571
C04181=1034.855,0.474,-86.574,168.667,40.452,157.571
C04182=1034.861,0.724,-86.589,168.670,40.452,157.571
C04183=1034.867,0.973,-86.603,168.672,40.452,157.571
C04184=1034.873,1.222,-86.618,168.675,40.451,157.571
C04185=1034.880,1.472,-86.633,168.678,40.451,157.571
C04186=1034.886,1.722,-86.648,168.680,40.451,157.571
C04187=1034.892,1.971,-86.663,168.681,40.450,157.571
C04188=1034.899,2.220,-86.679,168.684,40.450,157.571
C04189=1034.905,2.469,-86.693,168.687,40.450,157.571
C04190=1034.911,2.719,-86.708,168.689,40.449,157.571
C04191=1034.918,2.968,-86.723,168.691,40.449,157.571
C04192=1034.924,3.218,-86.738,168.693,40.448,157.571
C04193=1034.930,3.468,-86.753,168.695,40.448,157.571
C04194=1034.936,3.717,-86.768,168.697,40.448,157.571
C04195=1034.942,3.966,-86.782,168.701,40.447,157.572
C04196=1034.948,4.216,-86.798,168.703,40.447,157.572
C04197=1034.955,4.465,-86.814,168.704,40.446,157.572
C04198=1034.961,4.715,-86.829,168.706,40.446,157.572
C04199=1034.968,4.965,-86.844,168.709,40.446,157.572
C04200=1034.973,5.214,-86.858,168.712,40.446,157.572
C04201=1034.980,5.463,-86.873,168.714,40.446,157.572
C04202=1034.986,5.713,-86.888,168.716,40.445,157.572
C04203=1034.993,5.962,-86.904,168.718,40.444,157.572
C04204=1034.999,6.212,-86.919,168.720,40.444,157.572
C04205=1035.006,6.461,-86.934,168.723,40.444,157.572
C04206=1035.012,6.711,-86.949,168.726,40.444,157.572
C04207=1035.018,6.961,-86.963,168.727,40.443,157.572
C04208=1035.025,7.210,-86.979,168.729,40.443,157.572
C04209=1035.031,7.459,-86.994,168.732,40.442,157.572
C04210=1035.037,7.708,-87.009,168.734,40.442,157.572
C04211=1035.044,7.958,-87.024,168.736,40.441,157.572
C04212=1035.050,8.207,-87.039,168.738,40.441,157.572
C04213=1035.057,8.457,-87.054,168.741,40.441,157.572
C04214=1035.063,8.706,-87.069,168.743,40.440,157.572
C04215=1035.069,8.956,-87.084,168.745,40.440,157.572
C04216=1035.076,9.205,-87.100,168.748,40.439,157.572
C04217=1035.082,9.455,-87.115,168.750,40.439,157.572
C04218=1035.088,9.705,-87.130,168.752,40.439,157.572
C04219=1035.094,9.954,-87.145,168.754,40.439,157.572
C04220=1035.101,10.203,-87.161,168.757,40.438,157.572
C04221=1035.108,10.453,-87.176,168.759,40.438,157.572
C04222=1035.114,10.703,-87.191,168.761,40.437,157.572
C04223=1035.121,10.952,-87.206,168.764,40.437,157.573
C04224=1035.127,11.201,-87.221,168.766,40.436,157.572
C04225=1035.133,11.451,-87.236,168.768,40.436,157.572
C04226=1035.140,11.700,-87.252,168.770,40.436,157.573
C04227=1035.147,11.985,-87.269,168.773,40.435,157.573
C04228=1035.154,12.270,-87.286,168.776,40.434,157.573
C04229=1035.162,12.556,-87.304,168.778,40.434,157.573
C04230=1035.169,12.841,-87.322,168.781,40.434,157.573
C04231=1035.176,13.090,-87.337,168.783,40.434,157.573
C04232=1035.182,13.339,-87.352,168.785,40.433,157.573
C04233=1035.189,13.589,-87.367,168.788,40.433,157.573
C04234=1035.194,13.839,-87.383,168.790,40.432,157.573
C04235=1035.201,14.088,-87.398,168.792,40.432,157.573
C04236=1035.208,14.338,-87.413,168.794,40.431,157.573
C04237=1035.213,14.587,-87.430,168.797,40.431,157.573
C04238=1035.220,14.837,-87.445,168.799,40.431,157.573
C04239=1035.227,15.086,-87.460,168.801,40.431,157.573
C04240=1035.232,15.336,-87.476,168.803,40.430,157.573
C04241=1035.239,15.585,-87.491,168.806,40.430,157.573
C04242=1035.245,15.835,-87.506,168.808,40.430,157.573
C04243=1035.251,16.084,-87.523,168.810,40.430,157.573
C04244=1035.258,16.333,-87.538,168.812,40.430,157.573
C04245=1035.264,16.583,-87.553,168.814,40.429,157.573
C04246=1035.270,16.832,-87.569,168.817,40.428,157.573
C04247=1035.277,17.082,-87.584,168.819,40.428,157.573
C04248=1035.283,17.331,-87.600,168.821,40.428,157.573
C04249=1035.289,17.581,-87.616,168.823,40.428,157.573
C04250=1035.296,17.830,-87.632,168.826,40.427,157.574
C04251=1035.303,18.079,-87.647,168.828,40.427,157.574
C04252=1035.309,18.329,-87.663,168.830,40.427,157.574
C04253=1035.315,18.578,-87.678,168.832,40.426,157.574
C04254=1035.322,18.827,-87.694,168.834,40.426,157.574
C04255=1035.328,19.077,-87.710,168.837,40.426,157.574
C04256=1035.334,19.326,-87.725,168.839,40.425,157.574
C04257=1035.341,19.576,-87.740,168.841,40.425,157.574
C04258=1035.347,19.825,-87.757,168.843,40.425,157.574
C04259=1035.353,20.074,-87.772,168.845,40.425,157.574
C04260=1035.359,20.324,-87.788,168.849,40.425,157.574
C04261=1035.366,20.573,-87.803,168.851,40.424,157.574
C04262=1035.372,20.823,-87.820,168.852,40.423,157.574
C04263=1035.379,21.073,-87.836,168.854,40.423,157.574
C04264=1035.385,21.323,-87.851,168.856,40.423,157.574
C04265=1035.391,21.572,-87.867,168.859,40.423,157.574
C04266=1035.397,21.821,-87.883,168.862,40.423,157.574
C04267=1035.404,22.070,-87.899,168.864,40.422,157.574
C04268=1035.410,22.319,-87.915,168.866,40.422,157.574
C04269=1035.416,22.569,-87.930,168.868,40.422,157.574
C04270=1035.422,22.818,-87.946,168.871,40.422,157.574
C04271=1035.429,23.067,-87.962,168.873,40.421,157.574
C04272=1035.435,23.317,-87.979,168.875,40.421,157.575
C04273=1035.442,23.567,-87.994,168.877,40.421,157.575
C04274=1035.448,23.816,-88.010,168.879,40.421,157.575
C04275=1035.454,24.065,-88.025,168.882,40.420,157.575
C04276=1035.460,24.315,-88.042,168.884,40.420,157.575
C04277=1035.467,24.564,-88.057,168.886,40.419,157.575
C04278=1035.473,24.813,-88.074,168.888,40.419,157.575
C04279=1035.480,25.064,-88.089,168.890,40.419,157.575
C04280=1035.486,25.313,-88.105,168.893,40.419,157.575
C04281=1035.492,25.562,-88.121,168.895,40.419,157.575
C04282=1035.499,25.811,-88.137,168.897,40.418,157.575
C04283=1035.505,26.061,-88.153,168.899,40.418,157.575
C04284=1035.512,26.310,-88.169,168.901,40.418,157.575
C04285=1035.518,26.560,-88.186,168.904,40.417,157.575
C04286=1035.524,26.809,-88.201,168.906,40.417,157.575
C04287=1035.530,27.058,-88.218,168.908,40.417,157.575
C04288=1035.537,27.308,-88.232,168.910,40.416,157.575
C04289=1035.543,27.558,-88.249,168.912,40.416,157.575
C04290=1035.549,27.807,-88.265,168.914,40.416,157.575
C04291=1035.557,28.093,-88.284,168.917,40.416,157.575
C04292=1035.564,28.380,-88.303,168.919,40.415,157.575
C04293=1035.571,28.666,-88.321,168.922,40.415,157.575
C04294=1035.579,28.953,-88.339,168.924,40.415,157.576
C04295=1035.585,29.202,-88.355,168.927,40.415,157.576
C04296=1035.590,29.451,-88.372,168.929,40.414,157.576
C04297=1035.598,29.701,-88.388,168.931,40.414,157.576
C04298=1035.604,29.951,-88.404,168.933,40.414,157.576
C04299=1035.610,30.200,-88.420,168.935,40.414,157.576
C04300=1035.616,30.449,-88.437,168.937,40.414,157.576
C04301=1035.623,30.699,-88.453,168.939,40.413,157.576
C04302=1035.629,30.948,-88.469,168.942,40.413,157.576
C04303=1035.635,31.197,-88.486,168.944,40.413,157.576
C04304=1035.641,31.446,-88.502,168.946,40.413,157.576
C04305=1035.648,31.696,-88.518,168.948,40.413,157.576
C04306=1035.654,31.945,-88.534,168.950,40.412,157.576
C04307=1035.660,32.195,-88.551,168.952,40.412,157.576
C04308=1035.666,32.444,-88.567,168.955,40.412,157.576
C04309=1035.673,32.694,-88.583,168.957,40.412,157.576
C04310=1035.679,32.943,-88.599,168.959,40.411,157.576
C04311=1035.685,33.193,-88.615,168.961,40.411,157.577
C04312=1035.692,33.441,-88.632,168.963,40.411,157.577
C04313=1035.698,33.691,-88.649,168.965,40.411,157.577
C04314=1035.705,33.940,-88.665,168.967,40.410,157.577
C04315=1035.711,34.190,-88.681,168.970,40.410,157.577
C04316=1035.717,34.440,-88.698,168.972,40.409,157.577
C04317=1035.723,34.689,-88.714,168.974,40.409,157.577
C04318=1035.730,34.938,-88.730,168.976,40.409,157.577
C04319=1035.737,35.188,-88.747,168.978,40.409,157.577
C04320=1035.743,35.437,-88.763,168.980,40.409,157.577
C04321=1035.749,35.686,-88.779,168.982,40.408,157.577
C04322=1035.755,35.936,-88.796,168.985,40.408,157.577
C04323=1035.762,36.185,-88.812,168.988,40.408,157.577
C04324=1035.768,36.434,-88.829,168.990,40.408,157.577
C04325=1035.775,36.684,-88.845,168.992,40.407,157.577
C04326=1035.781,36.934,-88.861,168.994,40.407,157.577
C04327=1035.787,37.182,-88.878,168.996,40.407,157.577
C04328=1035.794,37.432,-88.894,168.999,40.407,157.577
C04329=1035.800,37.681,-88.911,169.001,40.407,157.577
C04330=1035.807,37.930,-88.928,169.003,40.406,157.577
C04331=1035.813,38.180,-88.944,169.005,40.406,157.578
C04332=1035.819,38.429,-88.961,169.007,40.406,157.578
C04333=1035.825,38.678,-88.977,169.009,40.406,157.578
C04334=1035.832,38.928,-88.994,169.011,40.406,157.578
C04335=1035.838,39.178,-89.010,169.013,40.405,157.578
C04336=1035.844,39.426,-89.027,169.015,40.405,157.578
C04337=1035.851,39.676,-89.044,169.018,40.405,157.578
C04338=1035.857,39.926,-89.060,169.020,40.405,157.578
C04339=1035.862,40.175,-89.078,169.022,40.404,157.578
C04340=1035.869,40.425,-89.094,169.024,40.404,157.578
C04341=1035.875,40.674,-89.111,169.026,40.404,157.578
C04342=1035.881,40.924,-89.128,169.028,40.404,157.578
C04343=1035.888,41.172,-89.145,169.030,40.404,157.578
C04344=1035.894,41.422,-89.161,169.032,40.404,157.578
C04345=1035.900,41.672,-89.178,169.035,40.404,157.578
C04346=1035.906,41.920,-89.195,169.037,40.404,157.578
C04347=1035.912,42.170,-89.211,169.039,40.403,157.579
C04348=1035.919,42.419,-89.228,169.041,40.403,157.579
C04349=1035.925,42.669,-89.245,169.043,40.403,157.579
C04350=1035.932,42.918,-89.262,169.045,40.403,157.579
C04351=1035.938,43.167,-89.278,169.047,40.403,157.579
C04352=1035.945,43.417,-89.296,169.049,40.402,157.579
C04353=1035.951,43.666,-89.312,169.051,40.402,157.579
C04354=1035.956,43.915,-89.329,169.053,40.402,157.579
C04355=1035.964,44.202,-89.348,169.057,40.402,157.579
C04356=1035.971,44.488,-89.368,169.059,40.402,157.579
C04357=1035.978,44.775,-89.388,169.062,40.402,157.579
C04358=1035.985,45.061,-89.407,169.064,40.402,157.579
C04359=1035.991,45.311,-89.424,169.066,40.401,157.579
C04360=1035.998,45.559,-89.441,169.068,40.401,157.579
C04361=1036.004,45.810,-89.458,169.070,40.402,157.580
C04362=1036.010,46.058,-89.475,169.072,40.401,157.580
C04363=1036.016,46.308,-89.492,169.074,40.401,157.580
C04364=1036.022,46.558,-89.510,169.076,40.401,157.580
C04365=1036.028,46.806,-89.527,169.078,40.401,157.580
C04366=1036.035,47.056,-89.543,169.081,40.400,157.580
C04367=1036.040,47.305,-89.561,169.083,40.400,157.580
C04368=1036.047,47.555,-89.578,169.085,40.401,157.580
C04369=1036.053,47.804,-89.594,169.087,40.401,157.580
C04370=1036.060,48.054,-89.612,169.089,40.400,157.580
C04371=1036.065,48.303,-89.629,169.091,40.400,157.580
C04372=1036.072,48.552,-89.647,169.093,40.400,157.580
C04373=1036.078,48.801,-89.663,169.095,40.400,157.580
C04374=1036.084,49.051,-89.681,169.097,40.400,157.580
C04375=1036.091,49.300,-89.698,169.099,40.399,157.580
C04376=1036.097,49.549,-89.714,169.102,40.400,157.581
C04377=1036.103,49.799,-89.732,169.104,40.400,157.581
C04378=1036.109,50.048,-89.749,169.106,40.399,157.581
C04379=1036.116,50.297,-89.766,169.109,40.399,157.581
C04380=1036.122,50.546,-89.782,169.111,40.399,157.581
C04381=1036.128,50.796,-89.800,169.113,40.399,157.581
C04382=1036.135,51.046,-89.818,169.115,40.398,157.581
C04383=1036.141,51.294,-89.835,169.117,40.398,157.581
C04384=1036.147,51.545,-89.852,169.119,40.398,157.581
C04385=1036.153,51.793,-89.869,169.121,40.398,157.581
C04386=1036.160,52.043,-89.886,169.123,40.398,157.581
C04387=1036.165,52.292,-89.904,169.125,40.398,157.581
C04388=1036.172,52.541,-89.921,169.127,40.398,157.581
C04389=1036.179,52.790,-89.938,169.129,40.398,157.581
C04390=1036.184,53.040,-89.955,169.131,40.397,157.581
C04391=1036.191,53.289,-89.972,169.134,40.397,157.582
C04392=1036.197,53.539,-89.990,169.136,40.397,157.582
C04393=1036.203,53.788,-90.007,169.138,40.397,157.582
C04394=1036.210,54.037,-90.025,169.140,40.397,157.582
C04395=1036.217,54.286,-90.042,169.142,40.396,157.582
C04396=1036.222,54.536,-90.059,169.144,40.397,157.582
C04397=1036.229,54.786,-90.076,169.146,40.397,157.582
C04398=1036.235,55.034,-90.093,169.148,40.396,157.582
C04399=1036.241,55.284,-90.111,169.150,40.396,157.582
C04400=1036.248,55.533,-90.128,169.152,40.396,157.582
C04401=1036.254,55.782,-90.145,169.154,40.396,157.582
C04402=1036.260,56.032,-90.163,169.157,40.395,157.582
C04403=1036.267,56.281,-90.180,169.159,40.395,157.582
C04404=1036.273,56.530,-90.198,169.161,40.395,157.582
C04405=1036.280,56.780,-90.215,169.164,40.395,157.582
C04406=1036.286,57.029,-90.232,169.166,40.395,157.582
C04407=1036.293,57.278,-90.250,169.168,40.394,157.583
C04408=1036.299,57.528,-90.267,169.170,40.394,157.583
C04409=1036.305,57.777,-90.284,169.172,40.394,157.583
C04410=1036.312,58.027,-90.301,169.174,40.394,157.583
C04411=1036.317,58.276,-90.319,169.176,40.394,157.583
C04412=1036.324,58.525,-90.336,169.178,40.393,157.583
C04413=1036.330,58.775,-90.354,169.181,40.393,157.583
C04414=1036.336,59.023,-90.371,169.183,40.393,157.583
C04415=1036.343,59.273,-90.388,169.185,40.393,157.583
C04416=1036.349,59.523,-90.406,169.187,40.393,157.583
C04417=1036.356,59.771,-90.423,169.189,40.393,157.583
C04418=1036.363,60.021,-90.441,169.191,40.393,157.583
C04419=1036.370,60.307,-90.461,169.193,40.393,157.583
C04420=1036.377,60.593,-90.482,169.196,40.392,157.583
C04421=1036.385,60.879,-90.502,169.198,40.392,157.583
C04422=1036.392,61.165,-90.522,169.201,40.392,157.583
C04423=1036.399,61.415,-90.539,169.203,40.392,157.584
C04424=1036.405,61.663,-90.556,169.205,40.391,157.584
C04425=1036.411,61.913,-90.574,169.207,40.391,157.584
C04426=1036.418,62.163,-90.592,169.209,40.391,157.584
C04427=1036.424,62.412,-90.609,169.211,40.391,157.584
C04428=1036.430,62.661,-90.626,169.213,40.391,157.584
C04429=1036.437,62.911,-90.644,169.215,40.390,157.584
C04430=1036.443,63.160,-90.662,169.218,40.390,157.584
C04431=1036.450,63.410,-90.679,169.220,40.390,157.584
C04432=1036.457,63.658,-90.697,169.222,40.390,157.584
C04433=1036.463,63.908,-90.715,169.224,40.389,157.584
C04434=1036.469,64.157,-90.733,169.226,40.389,157.584
C04435=1036.475,64.406,-90.750,169.228,40.389,157.584
C04436=1036.481,64.656,-90.768,169.230,40.389,157.584
C04437=1036.488,64.905,-90.786,169.232,40.389,157.584
C04438=1036.495,65.154,-90.804,169.235,40.389,157.584
C04439=1036.500,65.403,-90.821,169.237,40.389,157.585
C04440=1036.506,65.653,-90.839,169.239,40.389,157.585
C04441=1036.513,65.902,-90.857,169.241,40.388,157.585
C04442=1036.520,66.152,-90.875,169.243,40.388,157.585
C04443=1036.525,66.401,-90.893,169.245,40.388,157.585
C04444=1036.532,66.650,-90.911,169.248,40.388,157.585
C04445=1036.538,66.899,-90.929,169.250,40.388,157.585
C04446=1036.544,67.149,-90.946,169.252,40.388,157.585
C04447=1036.551,67.398,-90.963,169.254,40.388,157.585
C04448=1036.557,67.647,-90.982,169.256,40.388,157.585
C04449=1036.563,67.897,-91.000,169.258,40.387,157.585
C04450=1036.569,68.146,-91.018,169.260,40.387,157.585
C04451=1036.576,68.394,-91.036,169.262,40.387,157.585
C04452=1036.582,68.644,-91.054,169.264,40.387,157.585
C04453=1036.588,68.894,-91.072,169.266,40.387,157.586
C04454=1036.595,69.143,-91.090,169.268,40.387,157.586
C04455=1036.601,69.392,-91.107,169.270,40.387,157.586
C04456=1036.607,69.641,-91.126,169.272,40.387,157.586
C04457=1036.613,69.891,-91.144,169.274,40.386,157.586
C04458=1036.620,70.140,-91.162,169.276,40.387,157.586
C04459=1036.626,70.390,-91.180,169.279,40.387,157.586
C04460=1036.632,70.638,-91.197,169.281,40.386,157.586
C04461=1036.639,70.887,-91.216,169.284,40.386,157.586
C04462=1036.645,71.137,-91.234,169.286,40.386,157.586
C04463=1036.651,71.386,-91.253,169.288,40.386,157.586
C04464=1036.657,71.636,-91.270,169.290,40.386,157.586
C04465=1036.663,71.884,-91.289,169.292,40.386,157.586
C04466=1036.669,72.134,-91.307,169.294,40.386,157.586
C04467=1036.676,72.383,-91.325,169.296,40.386,157.587
C04468=1036.683,72.633,-91.343,169.298,40.386,157.587
C04469=1036.689,72.882,-91.361,169.300,40.386,157.587
C04470=1036.695,73.131,-91.379,169.302,40.386,157.587
C04471=1036.701,73.380,-91.398,169.304,40.385,157.587
C04472=1036.707,73.630,-91.415,169.306,40.385,157.587
C04473=1036.713,73.879,-91.434,169.308,40.386,157.587
C04474=1036.720,74.129,-91.452,169.310,40.385,157.587
C04475=1036.726,74.378,-91.471,169.312,40.385,157.587
C04476=1036.732,74.626,-91.488,169.314,40.385,157.587
C04477=1036.739,74.876,-91.506,169.316,40.385,157.587
C04478=1036.745,75.125,-91.525,169.319,40.385,157.587
C04479=1036.751,75.374,-91.543,169.321,40.385,157.587
C04480=1036.758,75.624,-91.562,169.324,40.385,157.588
C04481=1036.764,75.873,-91.579,169.326,40.384,157.588
C04482=1036.770,76.122,-91.598,169.328,40.384,157.588
C04483=1036.778,76.408,-91.619,169.330,40.384,157.588
C04484=1036.785,76.694,-91.640,169.332,40.385,157.588
C04485=1036.792,76.980,-91.660,169.335,40.384,157.588
C04486=1036.799,77.266,-91.682,169.337,40.384,157.588
C04487=1036.805,77.515,-91.701,169.339,40.384,157.588
C04488=1036.812,77.765,-91.719,169.341,40.384,157.588
C04489=1036.818,78.014,-91.737,169.343,40.384,157.588
C04490=1036.824,78.263,-91.756,169.345,40.384,157.588
C04491=1036.830,78.512,-91.774,169.347,40.384,157.588
C04492=1036.836,78.762,-91.792,169.349,40.384,157.589
C04493=1036.843,79.011,-91.811,169.351,40.384,157.589
C04494=1036.849,79.260,-91.829,169.353,40.384,157.589
C04495=1036.855,79.500,-91.847,169.355,40.383,157.589
C04496=1036.860,79.739,-91.865,169.358,40.384,157.589
C04497=1036.867,79.979,-91.883,169.360,40.384,157.589
C04498=1036.872,80.218,-91.901,169.362,40.384,157.589
C04499=1036.878,80.458,-91.919,169.364,40.383,157.589
C04500=1036.885,80.697,-91.937,169.366,40.384,157.589
C04501=1036.890,80.936,-91.954,169.368,40.384,157.589
C04502=1036.896,81.177,-91.972,169.370,40.383,157.589
C04503=1036.903,81.426,-91.991,169.372,40.384,157.590
C04504=1036.909,81.675,-92.010,169.374,40.384,157.590
C04505=1036.915,81.924,-92.029,169.376,40.383,157.590
C04506=1036.921,82.173,-92.047,169.378,40.383,157.590
C04507=1036.927,82.423,-92.065,169.380,40.384,157.590
C04508=1036.934,82.672,-92.084,169.382,40.383,157.590
C04509=1036.940,82.921,-92.102,169.384,40.383,157.590
C04510=1036.945,83.170,-92.121,169.386,40.383,157.590
C04511=1036.952,83.419,-92.140,169.388,40.383,157.590
C04512=1036.958,83.668,-92.159,169.390,40.383,157.590
C04513=1036.965,83.917,-92.177,169.394,40.383,157.590
C04514=1036.971,84.166,-92.196,169.396,40.383,157.590
C04515=1036.977,84.417,-92.215,169.398,40.383,157.591
C04516=1036.983,84.666,-92.233,169.400,40.383,157.591
C04517=1036.989,84.915,-92.252,169.402,40.383,157.591
C04518=1036.996,85.164,-92.270,169.404,40.383,157.591
C04519=1037.002,85.413,-92.289,169.406,40.383,157.591
C04520=1037.009,85.662,-92.308,169.408,40.383,157.591
C04521=1037.014,85.912,-92.327,169.410,40.383,157.591
C04522=1037.021,86.161,-92.346,169.412,40.382,157.591
C04523=1037.027,86.410,-92.364,169.414,40.383,157.591
C04524=1037.034,86.659,-92.383,169.416,40.383,157.591
C04525=1037.040,86.908,-92.402,169.418,40.382,157.591
C04526=1037.046,87.158,-92.421,169.420,40.382,157.591
C04527=1037.052,87.407,-92.439,169.422,40.382,157.591
C04528=1037.059,87.656,-92.458,169.424,40.382,157.592
C04529=1037.065,87.905,-92.477,169.426,40.382,157.592
C04530=1037.072,88.155,-92.496,169.429,40.382,157.592
C04531=1037.078,88.404,-92.515,169.432,40.382,157.592
C04532=1037.084,88.653,-92.534,169.434,40.382,157.592
C04533=1037.091,88.902,-92.552,169.436,40.382,157.592
C04534=1037.097,89.152,-92.571,169.438,40.382,157.592
C04535=1037.103,89.401,-92.590,169.440,40.382,157.592
C04536=1037.109,89.650,-92.609,169.442,40.381,157.592
C04537=1037.116,89.899,-92.628,169.444,40.382,157.592
C04538=1037.122,90.148,-92.646,169.446,40.382,157.592
C04539=1037.128,90.398,-92.665,169.448,40.381,157.592
C04540=1037.134,90.646,-92.685,169.450,40.382,157.593
C04541=1037.140,90.896,-92.704,169.452,40.382,157.593
C04542=1037.146,91.145,-92.723,169.454,40.381,157.593
C04543=1037.152,91.394,-92.742,169.456,40.382,157.593
C04544=1037.159,91.643,-92.761,169.458,40.382,157.593
C04545=1037.165,91.892,-92.781,169.460,40.381,157.593
C04546=1037.171,92.141,-92.799,169.463,40.382,157.593
C04547=1037.179,92.447,-92.823,169.466,40.382,157.593
C04548=1037.186,92.752,-92.846,169.468,40.382,157.593
C04549=1037.194,93.058,-92.869,169.471,40.382,157.594
C04550=1037.201,93.363,-92.893,169.473,40.382,157.594
C04551=1037.207,93.612,-92.912,169.475,40.382,157.594
C04552=1037.214,93.861,-92.931,169.478,40.382,157.594
C04553=1037.220,94.110,-92.951,169.480,40.381,157.594
C04554=1037.226,94.359,-92.969,169.482,40.382,157.594
C04555=1037.232,94.609,-92.989,169.484,40.382,157.594
C04556=1037.239,94.859,-93.008,169.486,40.381,157.594
C04557=1037.245,95.107,-93.028,169.488,40.382,157.594
C04558=1037.251,95.356,-93.046,169.490,40.382,157.594
C04559=1037.257,95.606,-93.066,169.492,40.382,157.594
C04560=1037.264,95.854,-93.085,169.495,40.382,157.595
C04561=1037.269,96.104,-93.104,169.497,40.382,157.595
C04562=1037.276,96.353,-93.123,169.499,40.382,157.595
C04563=1037.282,96.602,-93.143,169.501,40.381,157.595
C04564=1037.289,96.852,-93.162,169.503,40.382,157.595
C04565=1037.294,97.101,-93.181,169.505,40.382,157.595
C04566=1037.301,97.349,-93.200,169.507,40.381,157.595
C04567=1037.307,97.599,-93.220,169.509,40.382,157.595
C04568=1037.313,97.848,-93.238,169.511,40.382,157.595
C04569=1037.320,98.098,-93.259,169.514,40.381,157.595
C04570=1037.326,98.347,-93.277,169.516,40.382,157.596
C04571=1037.332,98.595,-93.297,169.518,40.382,157.596
C04572=1037.339,98.845,-93.316,169.520,40.381,157.596
C04573=1037.344,99.094,-93.335,169.522,40.381,157.596
C04574=1037.352,99.343,-93.355,169.525,40.382,157.596
C04575=1037.357,99.593,-93.374,169.527,40.381,157.596
C04576=1037.364,99.841,-93.393,169.529,40.381,157.596
C04577=1037.370,100.091,-93.413,169.531,40.382,157.596
C04578=1037.375,100.340,-93.432,169.533,40.381,157.596
C04579=1037.383,100.589,-93.452,169.535,40.381,157.596
C04580=1037.388,100.839,-93.471,169.537,40.382,157.596
C04581=1037.394,101.088,-93.491,169.539,40.381,157.596
C04582=1037.400,101.336,-93.511,169.541,40.382,157.597
C04583=1037.407,101.585,-93.530,169.543,40.382,157.597
C04584=1037.413,101.834,-93.549,169.546,40.381,157.597
C04585=1037.419,102.084,-93.569,169.548,40.382,157.597
C04586=1037.425,102.333,-93.589,169.550,40.382,157.597
C04587=1037.431,102.583,-93.608,169.553,40.382,157.597
C04588=1037.438,102.831,-93.628,169.555,40.382,157.597
C04589=1037.444,103.080,-93.648,169.557,40.382,157.597
C04590=1037.450,103.330,-93.667,169.559,40.382,157.597
C04591=1037.456,103.579,-93.687,169.561,40.382,157.597
C04592=1037.462,103.828,-93.706,169.563,40.382,157.598
C04593=1037.468,104.077,-93.726,169.565,40.382,157.598
C04594=1037.475,104.326,-93.746,169.567,40.382,157.598
C04595=1037.481,104.576,-93.765,169.569,40.382,157.598
C04596=1037.487,104.825,-93.785,169.571,40.382,157.598
C04597=1037.492,105.074,-93.805,169.573,40.383,157.598
C04598=1037.500,105.323,-93.824,169.575,40.382,157.598
C04599=1037.506,105.572,-93.844,169.578,40.383,157.598
C04600=1037.511,105.821,-93.863,169.581,40.382,157.598
C04601=1037.517,106.070,-93.883,169.583,40.382,157.599
C04602=1037.524,106.320,-93.904,169.585,40.383,157.599
C04603=1037.530,106.569,-93.922,169.587,40.382,157.599
C04604=1037.536,106.818,-93.942,169.589,40.382,157.599
C04605=1037.542,107.067,-93.962,169.591,40.383,157.599
C04606=1037.549,107.316,-93.983,169.593,40.383,157.599
C04607=1037.555,107.565,-94.002,169.595,40.383,157.599
C04608=1037.561,107.814,-94.021,169.597,40.383,157.599
C04609=1037.568,108.064,-94.042,169.599,40.383,157.599
C04610=1037.574,108.312,-94.062,169.601,40.383,157.600
C04611=1037.581,108.598,-94.084,169.604,40.383,157.600
C04612=1037.588,108.884,-94.107,169.607,40.383,157.600
C04613=1037.595,109.170,-94.130,169.610,40.383,157.600
C04614=1037.602,109.456,-94.152,169.612,40.383,157.600
C04615=1037.609,109.705,-94.172,169.614,40.383,157.600
C04616=1037.614,109.955,-94.192,169.616,40.383,157.600
C04617=1037.620,110.204,-94.212,169.618,40.383,157.600
C04618=1037.628,110.453,-94.231,169.620,40.383,157.600
C04619=1037.634,110.702,-94.251,169.623,40.383,157.600
C04620=1037.640,110.951,-94.272,169.625,40.383,157.601
C04621=1037.646,111.200,-94.292,169.627,40.383,157.601
C04622=1037.652,111.449,-94.311,169.629,40.383,157.601
C04623=1037.659,111.699,-94.331,169.631,40.383,157.601
C04624=1037.665,111.948,-94.351,169.634,40.383,157.601
C04625=1037.671,112.196,-94.371,169.636,40.383,157.601
C04626=1037.677,112.446,-94.391,169.638,40.383,157.601
C04627=1037.683,112.695,-94.411,169.640,40.384,157.601
C04628=1037.689,112.944,-94.431,169.642,40.383,157.601
C04629=1037.696,113.193,-94.452,169.644,40.384,157.602
C04630=1037.702,113.442,-94.472,169.647,40.384,157.602
C04631=1037.707,113.691,-94.492,169.649,40.384,157.602
C04632=1037.714,113.941,-94.513,169.651,40.384,157.602
C04633=1037.720,114.189,-94.532,169.653,40.384,157.602
C04634=1037.726,114.438,-94.552,169.655,40.384,157.602
C04635=1037.731,114.688,-94.573,169.658,40.384,157.602
C04636=1037.737,114.937,-94.593,169.660,40.385,157.602
C04637=1037.743,115.186,-94.613,169.662,40.385,157.603
C04638=1037.750,115.435,-94.634,169.664,40.385,157.603
C04639=1037.755,115.684,-94.654,169.666,40.385,157.603
C04640=1037.762,115.934,-94.674,169.668,40.385,157.603
C04641=1037.768,116.183,-94.694,169.670,40.385,157.603
C04642=1037.774,116.431,-94.714,169.672,40.386,157.603
C04643=1037.780,116.681,-94.735,169.675,40.386,157.603
C04644=1037.786,116.930,-94.755,169.677,40.386,157.603
C04645=1037.792,117.178,-94.776,169.680,40.386,157.604
C04646=1037.799,117.428,-94.796,169.682,40.386,157.604
C04647=1037.804,117.677,-94.817,169.684,40.386,157.604
C04648=1037.810,117.926,-94.837,169.686,40.386,157.604
C04649=1037.816,118.175,-94.857,169.688,40.387,157.604
C04650=1037.822,118.424,-94.878,169.690,40.386,157.604
C04651=1037.828,118.674,-94.898,169.692,40.387,157.604
C04652=1037.835,118.922,-94.919,169.694,40.387,157.604
C04653=1037.841,119.172,-94.939,169.697,40.387,157.605
C04654=1037.846,119.421,-94.960,169.699,40.388,157.605
C04655=1037.853,119.670,-94.980,169.702,40.387,157.605
C04656=1037.859,119.919,-95.000,169.704,40.388,157.605
C04657=1037.865,120.167,-95.020,169.706,40.387,157.605
C04658=1037.871,120.417,-95.041,169.708,40.388,157.605
C04659=1037.877,120.666,-95.061,169.710,40.388,157.605
C04660=1037.884,120.915,-95.082,169.712,40.388,157.605
C04661=1037.889,121.164,-95.102,169.714,40.388,157.605
C04662=1037.896,121.413,-95.123,169.716,40.388,157.606
C04663=1037.902,121.662,-95.143,169.719,40.388,157.606
C04664=1037.909,121.912,-95.164,169.722,40.388,157.606
C04665=1037.914,122.160,-95.185,169.724,40.388,157.606
C04666=1037.921,122.410,-95.205,169.726,40.389,157.606
C04667=1037.927,122.659,-95.225,169.728,40.388,157.606
C04668=1037.933,122.908,-95.246,169.730,40.389,157.606
C04669=1037.939,123.157,-95.267,169.732,40.389,157.607
C04670=1037.945,123.406,-95.287,169.734,40.389,157.607
C04671=1037.951,123.655,-95.308,169.736,40.390,157.607
C04672=1037.958,123.904,-95.329,169.739,40.389,157.607
C04673=1037.964,124.153,-95.349,169.742,40.390,157.607
C04674=1037.970,124.402,-95.369,169.744,40.389,157.607
C04675=1037.976,124.688,-95.393,169.746,40.390,157.607
C04676=1037.983,124.974,-95.417,169.749,40.390,157.607
C04677=1037.991,125.260,-95.441,169.751,40.390,157.607
C04678=1037.998,125.546,-95.464,169.754,40.390,157.608
C04679=1038.005,125.795,-95.485,169.756,40.390,157.608
C04680=1038.011,126.043,-95.505,169.758,40.390,157.608
C04681=1038.017,126.293,-95.526,169.760,40.390,157.608
C04682=1038.023,126.541,-95.546,169.762,40.390,157.608
C04683=1038.029,126.791,-95.567,169.765,40.391,157.608
C04684=1038.036,127.040,-95.588,169.768,40.390,157.608
C04685=1038.042,127.289,-95.608,169.770,40.391,157.608
C04686=1038.048,127.538,-95.629,169.772,40.391,157.609
C04687=1038.054,127.787,-95.649,169.774,40.391,157.609
C04688=1038.061,128.036,-95.671,169.776,40.391,157.609
C04689=1038.067,128.285,-95.691,169.778,40.391,157.609
C04690=1038.074,128.533,-95.712,169.781,40.391,157.609
C04691=1038.079,128.783,-95.733,169.783,40.391,157.609
C04692=1038.085,129.032,-95.753,169.785,40.391,157.609
C04693=1038.092,129.281,-95.774,169.788,40.392,157.609
C04694=1038.098,129.531,-95.795,169.790,40.391,157.609
C04695=1038.104,129.779,-95.815,169.793,40.392,157.610
C04696=1038.111,130.029,-95.836,169.795,40.391,157.610
C04697=1038.117,130.278,-95.857,169.797,40.392,157.610
C04698=1038.124,130.526,-95.878,169.799,40.392,157.610
C04699=1038.130,130.775,-95.898,169.801,40.392,157.610
C04700=1038.136,131.025,-95.920,169.803,40.392,157.610
C04701=1038.142,131.274,-95.941,169.806,40.392,157.610
C04702=1038.148,131.523,-95.962,169.809,40.393,157.611
C04703=1038.154,131.773,-95.983,169.811,40.392,157.611
C04704=1038.160,132.021,-96.004,169.813,40.393,157.611
C04705=1038.167,132.270,-96.025,169.815,40.393,157.611
C04706=1038.172,132.519,-96.045,169.817,40.393,157.611
C04707=1038.179,132.768,-96.066,169.820,40.393,157.611
C04708=1038.185,133.017,-96.088,169.822,40.394,157.611
C04709=1038.191,133.266,-96.109,169.824,40.394,157.611
C04710=1038.197,133.515,-96.130,169.826,40.394,157.612
C04711=1038.203,133.764,-96.151,169.829,40.395,157.612
C04712=1038.209,134.013,-96.173,169.831,40.394,157.612
C04713=1038.216,134.262,-96.193,169.834,40.395,157.612
C04714=1038.222,134.512,-96.215,169.836,40.395,157.612
C04715=1038.227,134.760,-96.236,169.838,40.395,157.612
C04716=1038.234,135.009,-96.257,169.840,40.395,157.612
C04717=1038.240,135.259,-96.278,169.842,40.396,157.613
C04718=1038.246,135.507,-96.299,169.844,40.396,157.613
C04719=1038.252,135.756,-96.320,169.848,40.396,157.613
C04720=1038.259,136.005,-96.342,169.850,40.396,157.613
C04721=1038.264,136.254,-96.363,169.852,40.396,157.613
C04722=1038.271,136.503,-96.383,169.854,40.397,157.613
C04723=1038.277,136.753,-96.405,169.856,40.396,157.613
C04724=1038.283,137.002,-96.427,169.859,40.397,157.614
C04725=1038.289,137.250,-96.447,169.861,40.397,157.614
C04726=1038.296,137.499,-96.469,169.863,40.397,157.614
C04727=1038.301,137.749,-96.490,169.865,40.397,157.614
C04728=1038.307,137.998,-96.511,169.868,40.398,157.614
C04729=1038.314,138.246,-96.532,169.871,40.397,157.614
C04730=1038.320,138.496,-96.554,169.873,40.398,157.614
C04731=1038.326,138.745,-96.575,169.875,40.398,157.615
C04732=1038.332,138.993,-96.597,169.877,40.399,157.615
C04733=1038.339,139.242,-96.618,169.879,40.399,157.615
C04734=1038.345,139.492,-96.639,169.882,40.399,157.615
C04735=1038.351,139.741,-96.661,169.885,40.399,157.615
C04736=1038.357,139.989,-96.682,169.887,40.399,157.615
C04737=1038.363,140.238,-96.704,169.889,40.399,157.615
C04738=1038.369,140.488,-96.726,169.891,40.400,157.616
C04739=1038.375,140.773,-96.750,169.894,40.400,157.616
C04740=1038.383,141.059,-96.775,169.896,40.401,157.616
C04741=1038.389,141.345,-96.799,169.899,40.401,157.616
C04742=1038.397,141.630,-96.824,169.902,40.401,157.616
C04743=1038.403,141.878,-96.845,169.905,40.401,157.616
C04744=1038.409,142.128,-96.866,169.907,40.402,157.617
C04745=1038.415,142.377,-96.888,169.909,40.402,157.617
C04746=1038.421,142.626,-96.910,169.911,40.402,157.617
C04747=1038.427,142.875,-96.931,169.913,40.402,157.617
C04748=1038.433,143.124,-96.953,169.916,40.403,157.617
C04749=1038.439,143.373,-96.974,169.919,40.403,157.617
C04750=1038.446,143.622,-96.997,169.921,40.403,157.617
C04751=1038.452,143.871,-97.018,169.923,40.403,157.618
C04752=1038.457,144.119,-97.039,169.926,40.403,157.618
C04753=1038.464,144.369,-97.061,169.928,40.404,157.618
C04754=1038.470,144.618,-97.083,169.930,40.404,157.618
C04755=1038.476,144.867,-97.104,169.932,40.404,157.618
C04756=1038.483,145.116,-97.125,169.935,40.404,157.618
C04757=1038.489,145.365,-97.147,169.938,40.405,157.619
C04758=1038.495,145.613,-97.169,169.940,40.405,157.619
C04759=1038.501,145.862,-97.191,169.942,40.405,157.619
C04760=1038.507,146.111,-97.212,169.944,40.406,157.619
C04761=1038.513,146.361,-97.234,169.947,40.406,157.619
C04762=1038.519,146.610,-97.256,169.949,40.406,157.619
C04763=1038.526,146.859,-97.277,169.951,40.406,157.620
C04764=1038.532,147.108,-97.300,169.954,40.407,157.620
C04765=1038.538,147.357,-97.321,169.957,40.407,157.620
C04766=1038.544,147.605,-97.342,169.959,40.407,157.620
C04767=1038.550,147.854,-97.364,169.961,40.408,157.620
C04768=1038.556,148.103,-97.387,169.963,40.407,157.620
C04769=1038.562,148.353,-97.409,169.966,40.408,157.621
C04770=1038.568,148.602,-97.430,169.968,40.408,157.621
C04771=1038.575,148.850,-97.453,169.971,40.409,157.621
C04772=1038.581,149.100,-97.474,169.973,40.409,157.621
C04773=1038.587,149.349,-97.496,169.976,40.409,157.621
C04774=1038.593,149.597,-97.518,169.978,40.409,157.621
C04775=1038.599,149.846,-97.540,169.980,40.410,157.621
C04776=1038.604,150.095,-97.562,169.982,40.410,157.622
C04777=1038.611,150.344,-97.584,169.986,40.410,157.622
C04778=1038.617,150.593,-97.606,169.988,40.411,157.622
C04779=1038.623,150.842,-97.628,169.990,40.411,157.622
C04780=1038.630,151.091,-97.650,169.993,40.412,157.622
C04781=1038.635,151.340,-97.672,169.995,40.412,157.623
C04782=1038.641,151.589,-97.694,169.997,40.412,157.623
C04783=1038.648,151.838,-97.716,169.999,40.412,157.623
C04784=1038.654,152.087,-97.738,170.003,40.413,157.623
C04785=1038.660,152.335,-97.760,170.005,40.413,157.623
C04786=1038.665,152.584,-97.783,170.007,40.413,157.623
C04787=1038.672,152.833,-97.804,170.009,40.414,157.624
C04788=1038.678,153.083,-97.826,170.012,40.414,157.624
C04789=1038.684,153.331,-97.848,170.014,40.415,157.624
C04790=1038.690,153.580,-97.870,170.016,40.414,157.624
C04791=1038.696,153.829,-97.893,170.020,40.415,157.624
C04792=1038.702,154.079,-97.914,170.022,40.415,157.624
C04793=1038.709,154.327,-97.937,170.024,40.416,157.625
C04794=1038.715,154.576,-97.958,170.026,40.416,157.625
C04795=1038.721,154.825,-97.981,170.029,40.416,157.625
C04796=1038.727,155.074,-98.004,170.032,40.417,157.625
C04797=1038.733,155.323,-98.026,170.034,40.417,157.625
C04798=1038.739,155.572,-98.048,170.037,40.417,157.626
C04799=1038.745,155.821,-98.070,170.039,40.418,157.626
C04800=1038.751,156.070,-98.093,170.041,40.418,157.626
C04801=1038.757,156.319,-98.115,170.043,40.419,157.626
C04802=1038.764,156.568,-98.137,170.047,40.419,157.626
C04803=1038.771,156.853,-98.163,170.049,40.419,157.626
C04804=1038.778,157.138,-98.188,170.052,40.420,157.627
C04805=1038.784,157.424,-98.214,170.055,40.420,157.627
C04806=1038.791,157.709,-98.239,170.057,40.421,157.627
C04807=1038.797,157.957,-98.262,170.060,40.421,157.627
C04808=1038.804,158.206,-98.284,170.063,40.421,157.627
C04809=1038.809,158.455,-98.306,170.065,40.422,157.628
C04810=1038.816,158.704,-98.329,170.068,40.422,157.628
C04811=1038.822,158.952,-98.351,170.070,40.422,157.628
C04812=1038.828,159.203,-98.374,170.072,40.423,157.628
C04813=1038.835,159.451,-98.396,170.076,40.423,157.628
C04814=1038.840,159.700,-98.419,170.078,40.424,157.629
C04815=1038.847,159.949,-98.441,170.080,40.424,157.629
C04816=1038.853,160.198,-98.463,170.083,40.424,157.629
C04817=1038.859,160.447,-98.486,170.085,40.425,157.629
C04818=1038.865,160.696,-98.509,170.087,40.425,157.629
C04819=1038.870,160.945,-98.532,170.090,40.426,157.630
C04820=1038.876,161.194,-98.555,170.093,40.426,157.630
C04821=1038.882,161.442,-98.577,170.095,40.427,157.630
C04822=1038.888,161.691,-98.600,170.097,40.427,157.630
C04823=1038.894,161.940,-98.623,170.100,40.428,157.630
C04824=1038.899,162.189,-98.645,170.103,40.428,157.631
C04825=1038.906,162.438,-98.668,170.105,40.429,157.631
C04826=1038.912,162.687,-98.691,170.108,40.429,157.631
C04827=1038.917,162.936,-98.713,170.110,40.430,157.631
C04828=1038.923,163.185,-98.736,170.112,40.430,157.632
C04829=1038.929,163.434,-98.759,170.115,40.431,157.632
C04830=1038.935,163.682,-98.782,170.118,40.431,157.632
C04831=1038.941,163.931,-98.805,170.120,40.432,157.632
C04832=1038.947,164.180,-98.828,170.122,40.433,157.632
C04833=1038.952,164.429,-98.851,170.125,40.433,157.633
C04834=1038.959,164.679,-98.874,170.128,40.433,157.633
C04835=1038.965,164.927,-98.896,170.130,40.434,157.633
C04836=1038.971,165.176,-98.919,170.133,40.434,157.633
C04837=1038.977,165.425,-98.942,170.135,40.435,157.633
C04838=1038.982,165.674,-98.965,170.137,40.436,157.634
C04839=1038.988,165.922,-98.989,170.141,40.436,157.634
C04840=1038.995,166.171,-99.011,170.143,40.436,157.634
C04841=1039.001,166.420,-99.034,170.145,40.437,157.634
C04842=1039.006,166.668,-99.057,170.148,40.437,157.634
C04843=1039.013,166.918,-99.080,170.151,40.438,157.635
C04844=1039.018,167.167,-99.103,170.154,40.438,157.635
C04845=1039.025,167.416,-99.126,170.156,40.439,157.635
C04846=1039.031,167.664,-99.149,170.158,40.439,157.635
C04847=1039.036,167.913,-99.171,170.161,40.440,157.636
C04848=1039.042,168.162,-99.195,170.164,40.441,157.636
C04849=1039.049,168.411,-99.218,170.166,40.441,157.636
C04850=1039.055,168.660,-99.241,170.169,40.441,157.636
C04851=1039.061,168.909,-99.264,170.171,40.442,157.636
C04852=1039.067,169.158,-99.287,170.173,40.442,157.637
C04853=1039.072,169.406,-99.310,170.177,40.443,157.637
C04854=1039.079,169.655,-99.334,170.179,40.444,157.637
C04855=1039.085,169.904,-99.357,170.182,40.444,157.637
C04856=1039.091,170.153,-99.379,170.184,40.444,157.638
C04857=1039.097,170.402,-99.402,170.186,40.445,157.638
C04858=1039.103,170.650,-99.426,170.190,40.446,157.638
C04859=1039.109,170.900,-99.449,170.192,40.446,157.638
C04860=1039.115,171.149,-99.472,170.195,40.446,157.638
C04861=1039.121,171.397,-99.495,170.197,40.447,157.639
C04862=1039.128,171.645,-99.518,170.199,40.448,157.639
C04863=1039.134,171.895,-99.541,170.203,40.448,157.639
C04864=1039.140,172.144,-99.564,170.205,40.449,157.639
C04865=1039.145,172.393,-99.587,170.208,40.449,157.640
C04866=1039.151,172.641,-99.611,170.210,40.450,157.640
C04867=1039.159,172.926,-99.637,170.214,40.450,157.640
C04868=1039.166,173.211,-99.664,170.217,40.451,157.640
C04869=1039.173,173.496,-99.690,170.220,40.452,157.641
C04870=1039.180,173.780,-99.717,170.222,40.452,157.641
C04871=1039.186,174.029,-99.740,170.225,40.452,157.641
C04872=1039.191,174.278,-99.763,170.228,40.453,157.641
C04873=1039.199,174.527,-99.786,170.231,40.454,157.641
C04874=1039.204,174.776,-99.809,170.233,40.454,157.642
C04875=1039.210,175.024,-99.833,170.236,40.454,157.642
C04876=1039.217,175.274,-99.856,170.239,40.456,157.642
C04877=1039.223,175.523,-99.879,170.241,40.456,157.642
C04878=1039.229,175.771,-99.903,170.244,40.456,157.643
C04879=1039.235,176.020,-99.926,170.246,40.457,157.643
C04880=1039.241,176.269,-99.950,170.249,40.458,157.643
C04881=1039.248,176.518,-99.973,170.252,40.458,157.643
C04882=1039.254,176.766,-99.996,170.255,40.458,157.643
C04883=1039.260,177.015,-100.019,170.257,40.459,157.644
C04884=1039.266,177.264,-100.043,170.260,40.460,157.644
C04885=1039.272,177.513,-100.066,170.262,40.460,157.644
C04886=1039.279,177.762,-100.090,170.266,40.460,157.644
C04887=1039.284,178.011,-100.113,170.268,40.461,157.645
C04888=1039.291,178.259,-100.137,170.271,40.462,157.645
C04889=1039.298,178.508,-100.160,170.273,40.462,157.645
C04890=1039.304,178.757,-100.183,170.277,40.463,157.645
C04891=1039.310,179.006,-100.207,170.279,40.463,157.645
C04892=1039.316,179.255,-100.230,170.282,40.464,157.646
C04893=1039.323,179.504,-100.254,170.284,40.464,157.646
C04894=1039.328,179.753,-100.277,170.287,40.465,157.646
C04895=1039.334,180.001,-100.301,170.290,40.466,157.647
C04896=1039.341,180.250,-100.324,170.293,40.466,157.647
C04897=1039.347,180.499,-100.348,170.295,40.466,157.647
C04898=1039.353,180.748,-100.372,170.298,40.467,157.647
C04899=1039.360,180.996,-100.394,170.301,40.468,157.647
C04900=1039.367,181.245,-100.418,170.304,40.468,157.648
C04901=1039.373,181.493,-100.442,170.306,40.468,157.648
C04902=1039.379,181.743,-100.465,170.309,40.469,157.648
C04903=1039.385,181.991,-100.489,170.312,40.470,157.648
C04904=1039.392,182.240,-100.513,170.315,40.470,157.649
C04905=1039.397,182.489,-100.536,170.318,40.470,157.649
C04906=1039.404,182.738,-100.560,170.320,40.472,157.649
C04907=1039.410,182.986,-100.584,170.323,40.472,157.649
C04908=1039.416,183.236,-100.607,170.325,40.472,157.649
C04909=1039.422,183.484,-100.631,170.329,40.473,157.650
C04910=1039.429,183.733,-100.655,170.331,40.474,157.650
C04911=1039.435,183.982,-100.678,170.334,40.475,157.650
C04912=1039.441,184.231,-100.703,170.336,40.475,157.651
C04913=1039.447,184.479,-100.726,170.340,40.476,157.651
C04914=1039.453,184.728,-100.751,170.342,40.477,157.651
C04915=1039.459,184.977,-100.775,170.345,40.477,157.651
C04916=1039.465,185.226,-100.799,170.348,40.478,157.652
C04917=1039.471,185.474,-100.823,170.351,40.479,157.652
C04918=1039.476,185.723,-100.847,170.353,40.480,157.652
C04919=1039.483,185.972,-100.871,170.356,40.481,157.653
C04920=1039.488,186.220,-100.896,170.359,40.481,157.653
C04921=1039.495,186.469,-100.920,170.362,40.482,157.653
C04922=1039.500,186.718,-100.944,170.364,40.483,157.653
C04923=1039.507,186.967,-100.968,170.368,40.483,157.654
C04924=1039.512,187.216,-100.992,170.370,40.484,157.654
C04925=1039.519,187.465,-101.016,170.373,40.485,157.654
C04926=1039.524,187.713,-101.040,170.375,40.486,157.654
C04927=1039.531,187.962,-101.064,170.379,40.487,157.655
C04928=1039.536,188.211,-101.089,170.382,40.488,157.655
C04929=1039.542,188.460,-101.113,170.384,40.488,157.655
C04930=1039.548,188.709,-101.137,170.388,40.489,157.656
C04931=1039.555,188.993,-101.165,170.391,40.490,157.656
C04932=1039.562,189.277,-101.192,170.393,40.491,157.656
C04933=1039.570,189.562,-101.221,170.397,40.492,157.657
C04934=1039.576,189.846,-101.248,170.400,40.492,157.657
C04935=1039.582,190.095,-101.272,170.403,40.493,157.657
C04936=1039.588,190.343,-101.297,170.405,40.494,157.658
C04937=1039.594,190.592,-101.321,170.409,40.494,157.658
C04938=1039.601,190.841,-101.345,170.412,40.495,157.658
C04939=1039.606,191.090,-101.369,170.414,40.496,157.658
C04940=1039.613,191.339,-101.393,170.417,40.497,157.659
C04941=1039.618,191.586,-101.418,170.420,40.498,157.659
C04942=1039.625,191.835,-101.442,170.423,40.499,157.659
C04943=1039.631,192.085,-101.467,170.426,40.500,157.660
C04944=1039.637,192.333,-101.491,170.429,40.500,157.660
C04945=1039.643,192.582,-101.515,170.432,40.501,157.660
C04946=1039.650,192.831,-101.540,170.434,40.502,157.660
C04947=1039.655,193.079,-101.564,170.437,40.502,157.661
C04948=1039.662,193.328,-101.588,170.441,40.503,157.661
C04949=1039.668,193.577,-101.614,170.443,40.504,157.661
C04950=1039.673,193.825,-101.638,170.446,40.505,157.662
C04951=1039.680,194.074,-101.662,170.449,40.506,157.662
C04952=1039.686,194.323,-101.687,170.452,40.507,157.662
C04953=1039.692,194.571,-101.711,170.455,40.507,157.663
C04954=1039.698,194.821,-101.736,170.457,40.508,157.663
C04955=1039.705,195.069,-101.760,170.461,40.509,157.663
C04956=1039.711,195.318,-101.785,170.464,40.510,157.663
C04957=1039.717,195.567,-101.809,170.466,40.511,157.664
C04958=1039.723,195.815,-101.834,170.470,40.511,157.664
C04959=1039.730,196.064,-101.858,170.473,40.512,157.664
C04960=1039.735,196.312,-101.883,170.475,40.513,157.665
C04961=1039.742,196.561,-101.907,170.479,40.514,157.665
C04962=1039.748,196.811,-101.932,170.481,40.514,157.665
C04963=1039.754,197.059,-101.957,170.484,40.515,157.665
C04964=1039.760,197.307,-101.981,170.488,40.516,157.666
C04965=1039.766,197.556,-102.006,170.490,40.517,157.666
C04966=1039.773,197.805,-102.030,170.493,40.518,157.666
C04967=1039.779,198.054,-102.055,170.496,40.519,157.667
C04968=1039.786,198.303,-102.079,170.500,40.519,157.667
C04969=1039.791,198.551,-102.104,170.502,40.521,157.667
C04970=1039.797,198.800,-102.129,170.505,40.521,157.668
C04971=1039.804,199.048,-102.154,170.509,40.522,157.668
C04972=1039.810,199.298,-102.178,170.511,40.523,157.668
C04973=1039.817,199.546,-102.203,170.514,40.524,157.669
C04974=1039.823,199.795,-102.228,170.518,40.525,157.669
C04975=1039.829,200.043,-102.252,170.520,40.526,157.669
C04976=1039.835,200.292,-102.277,170.523,40.526,157.669
C04977=1039.841,200.541,-102.302,170.526,40.527,157.670
C04978=1039.848,200.789,-102.327,170.530,40.528,157.670
C04979=1039.855,201.038,-102.352,170.532,40.529,157.670
C04980=1039.860,201.287,-102.377,170.535,40.530,157.671
C04981=1039.867,201.536,-102.402,170.539,40.531,157.671
C04982=1039.872,201.784,-102.427,170.541,40.532,157.671
C04983=1039.879,202.033,-102.451,170.544,40.533,157.672
C04984=1039.885,202.282,-102.476,170.548,40.534,157.672
C04985=1039.891,202.530,-102.502,170.550,40.535,157.672
C04986=1039.897,202.779,-102.527,170.553,40.536,157.673
C04987=1039.904,203.028,-102.552,170.557,40.537,157.673
C04988=1039.909,203.276,-102.577,170.559,40.538,157.673
C04989=1039.915,203.525,-102.602,170.562,40.538,157.674
C04990=1039.921,203.773,-102.627,170.566,40.539,157.674
C04991=1039.928,204.022,-102.653,170.569,40.540,157.674
C04992=1039.934,204.271,-102.678,170.571,40.541,157.675
C04993=1039.940,204.519,-102.703,170.575,40.542,157.675
C04994=1039.946,204.769,-102.728,170.578,40.543,157.675
C04995=1039.972,205.819,-102.834,170.868,40.647,157.710
C04996=1039.981,206.126,-102.866,170.870,40.649,157.711
C04997=1039.989,206.433,-102.900,170.873,40.651,157.712
C04998=1039.997,206.740,-102.932,170.876,40.653,157.712
C04999=1040.006,207.047,-102.965,170.878,40.655,157.713
C05000=1040.013,207.296,-102.991,170.881,40.657,157.713
C05001=1040.019,207.544,-103.017,170.883,40.659,157.714
C05002=1040.026,207.793,-103.044,170.885,40.661,157.714
C05003=1040.032,208.041,-103.070,170.887,40.662,157.715
C05004=1040.039,208.290,-103.097,170.890,40.664,157.715
C05005=1040.045,208.537,-103.124,170.892,40.666,157.715
C05006=1040.052,208.786,-103.150,170.894,40.667,157.716
C05007=1040.059,209.035,-103.177,170.896,40.669,157.716
C05008=1040.065,209.283,-103.203,170.899,40.671,157.717
C05009=1040.072,209.532,-103.230,170.901,40.672,157.717
C05010=1040.079,209.781,-103.256,170.903,40.675,157.718
C05011=1040.085,210.029,-103.283,170.905,40.676,157.718
C05012=1040.092,210.278,-103.309,170.908,40.678,157.719
C05013=1040.099,210.525,-103.336,170.910,40.680,157.719
C05014=1040.106,210.774,-103.363,170.912,40.681,157.720
C05015=1040.113,211.023,-103.389,170.914,40.683,157.720
C05016=1040.119,211.271,-103.416,170.917,40.685,157.721
C05017=1040.126,211.520,-103.443,170.919,40.686,157.721
C05018=1040.133,211.768,-103.470,170.921,40.688,157.721
C05019=1040.139,212.017,-103.496,170.923,40.690,157.722
C05020=1040.146,212.265,-103.523,170.926,40.692,157.723
C05021=1040.152,212.514,-103.549,170.928,40.694,157.723
C05022=1040.158,212.762,-103.577,170.930,40.695,157.723
C05023=1040.165,213.011,-103.604,170.932,40.697,157.724
C05024=1040.171,213.259,-103.630,170.935,40.699,157.724
C05025=1040.179,213.508,-103.657,170.938,40.701,157.725
C05026=1040.185,213.757,-103.684,170.940,40.702,157.725
C05027=1040.191,214.005,-103.710,170.942,40.704,157.726
C05028=1040.198,214.253,-103.738,170.944,40.706,157.726
C05029=1040.205,214.502,-103.765,170.947,40.707,157.727
C05030=1040.211,214.750,-103.791,170.949,40.709,157.727
C05031=1040.218,214.998,-103.818,170.952,40.711,157.728
C05032=1040.225,215.247,-103.845,170.953,40.712,157.728
C05033=1040.231,215.495,-103.873,170.956,40.715,157.729
C05034=1040.238,215.744,-103.899,170.958,40.716,157.729
C05035=1040.244,215.993,-103.926,170.961,40.718,157.730
C05036=1040.252,216.241,-103.953,170.963,40.720,157.730
C05037=1040.258,216.489,-103.980,170.965,40.721,157.731
C05038=1040.265,216.738,-104.007,170.967,40.723,157.731
C05039=1040.271,216.987,-104.034,170.970,40.725,157.732
C05040=1040.278,217.235,-104.062,170.972,40.726,157.732
C05041=1040.285,217.483,-104.088,170.975,40.729,157.733
C05042=1040.291,217.732,-104.116,170.977,40.730,157.733
C05043=1040.298,217.980,-104.142,170.979,40.732,157.733
C05044=1040.305,218.229,-104.170,170.981,40.734,157.734
C05045=1040.312,218.477,-104.196,170.984,40.735,157.734
C05046=1040.318,218.725,-104.224,170.986,40.737,157.735
C05047=1040.325,218.974,-104.251,170.989,40.738,157.735
C05048=1040.332,219.222,-104.278,170.991,40.740,157.736
C05049=1040.338,219.471,-104.305,170.994,40.742,157.736
C05050=1040.345,219.719,-104.331,170.996,40.743,157.737
C05051=1040.352,219.968,-104.358,170.998,40.745,157.737
C05052=1040.360,220.280,-104.393,171.002,40.747,157.738
C05053=1040.368,220.593,-104.427,171.004,40.749,157.738
C05054=1040.376,220.906,-104.461,171.007,40.752,157.739
C05055=1040.385,221.218,-104.496,171.011,40.754,157.740
C05056=1040.391,221.467,-104.524,171.013,40.756,157.740
C05057=1040.397,221.714,-104.551,171.015,40.758,157.741
C05058=1040.405,221.963,-104.577,171.017,40.759,157.741
C05059=1040.411,222.211,-104.605,171.020,40.761,157.742
C05060=1040.418,222.460,-104.633,171.022,40.763,157.742
C05061=1040.425,222.708,-104.661,171.025,40.765,157.743
C05062=1040.430,222.957,-104.687,171.027,40.767,157.743
C05063=1040.437,223.205,-104.715,171.030,40.768,157.744
C05064=1040.445,223.453,-104.742,171.032,40.770,157.744
C05065=1040.451,223.702,-104.770,171.035,40.771,157.745
C05066=1040.458,223.951,-104.797,171.036,40.773,157.745
C05067=1040.464,224.199,-104.825,171.039,40.775,157.746
C05068=1040.471,224.448,-104.852,171.042,40.777,157.746
C05069=1040.477,224.695,-104.880,171.044,40.779,157.747
C05070=1040.484,224.944,-104.907,171.047,40.780,157.747
C05071=1040.491,225.192,-104.934,171.049,40.782,157.747
C05072=1040.497,225.441,-104.962,171.052,40.784,157.748
C05073=1040.504,225.689,-104.989,171.054,40.785,157.748
C05074=1040.511,225.938,-105.017,171.057,40.787,157.749
C05075=1040.518,226.186,-105.045,171.059,40.789,157.749
C05076=1040.524,226.435,-105.072,171.062,40.791,157.750
C05077=1040.530,226.683,-105.100,171.064,40.792,157.750
C05078=1040.537,226.931,-105.128,171.067,40.794,157.751
C05079=1040.544,227.179,-105.155,171.069,40.795,157.751
C05080=1040.551,227.428,-105.182,171.072,40.797,157.752
C05081=1040.557,227.677,-105.209,171.074,40.799,157.752
C05082=1040.564,227.925,-105.237,171.076,40.801,157.753
C05083=1040.571,228.174,-105.265,171.078,40.803,157.753
C05084=1040.577,228.422,-105.293,171.081,40.804,157.754
C05085=1040.584,228.670,-105.320,171.083,40.806,157.754
C05086=1040.591,228.919,-105.348,171.086,40.808,157.755
C05087=1040.598,229.167,-105.376,171.089,40.810,157.755
C05088=1040.604,229.416,-105.404,171.091,40.811,157.756
C05089=1040.611,229.664,-105.431,171.094,40.813,157.756
C05090=1040.618,229.912,-105.460,171.096,40.815,157.757
C05091=1040.624,230.160,-105.487,171.099,40.816,157.757
C05092=1040.630,230.408,-105.515,171.101,40.819,157.758
C05093=1040.637,230.657,-105.543,171.104,40.820,157.758
C05094=1040.643,230.905,-105.571,171.106,40.822,157.759
C05095=1040.650,231.154,-105.599,171.109,40.823,157.759
C05096=1040.657,231.402,-105.626,171.112,40.826,157.760
C05097=1040.663,231.651,-105.654,171.114,40.827,157.760
C05098=1040.670,231.899,-105.682,171.117,40.829,157.761
C05099=1040.677,232.147,-105.710,171.119,40.830,157.761
C05100=1040.683,232.396,-105.739,171.122,40.832,157.762
C05101=1040.690,232.644,-105.766,171.124,40.834,157.762
C05102=1040.696,232.893,-105.794,171.127,40.836,157.763
C05103=1040.703,233.140,-105.822,171.129,40.838,157.763
C05104=1040.709,233.389,-105.851,171.132,40.840,157.764
C05105=1040.716,233.638,-105.878,171.134,40.841,157.764
C05106=1040.723,233.886,-105.906,171.137,40.843,157.765
C05107=1040.730,234.134,-105.935,171.139,40.845,157.765
C05108=1040.738,234.440,-105.969,171.143,40.847,157.766
C05109=1040.745,234.744,-106.003,171.146,40.849,157.766
C05110=1040.754,235.049,-106.038,171.149,40.851,157.767
C05111=1040.762,235.355,-106.073,171.152,40.853,157.768
C05112=1040.769,235.603,-106.101,171.155,40.855,157.768
C05113=1040.776,235.851,-106.129,171.157,40.857,157.769
C05114=1040.781,236.100,-106.158,171.160,40.859,157.769
C05115=1040.788,236.348,-106.185,171.162,40.860,157.770
C05116=1040.795,236.596,-106.214,171.165,40.862,157.770
C05117=1040.802,236.844,-106.242,171.168,40.864,157.771
C05118=1040.808,237.093,-106.270,171.170,40.866,157.771
C05119=1040.815,237.341,-106.298,171.173,40.867,157.772
C05120=1040.821,237.589,-106.326,171.176,40.869,157.772
C05121=1040.828,237.837,-106.355,171.179,40.871,157.773
C05122=1040.834,238.086,-106.383,171.181,40.873,157.773
C05123=1040.841,238.334,-106.411,171.184,40.874,157.774
C05124=1040.849,238.583,-106.439,171.186,40.876,157.774
C05125=1040.855,238.831,-106.468,171.189,40.878,157.775
C05126=1040.862,239.079,-106.496,171.192,40.880,157.775
C05127=1040.868,239.328,-106.525,171.194,40.881,157.776
C05128=1040.874,239.576,-106.553,171.197,40.883,157.776
C05129=1040.881,239.824,-106.581,171.199,40.885,157.777
C05130=1040.887,240.073,-106.610,171.202,40.887,157.777
C05131=1040.894,240.320,-106.638,171.205,40.888,157.778
C05132=1040.902,240.570,-106.666,171.208,40.890,157.778
C05133=1040.908,240.818,-106.695,171.210,40.892,157.779
C05134=1040.915,241.066,-106.723,171.213,40.894,157.779
C05135=1040.921,241.314,-106.752,171.215,40.895,157.780
C05136=1040.928,241.562,-106.781,171.218,40.898,157.780
C05137=1040.934,241.810,-106.810,171.221,40.899,157.781
C05138=1040.941,242.059,-106.837,171.223,40.901,157.781
C05139=1040.948,242.308,-106.867,171.226,40.903,157.782
C05140=1040.955,242.555,-106.895,171.228,40.905,157.782
C05141=1040.961,242.804,-106.923,171.232,40.906,157.783
C05142=1040.967,243.052,-106.952,171.235,40.908,157.784
C05143=1040.974,243.300,-106.981,171.237,40.910,157.784
C05144=1040.980,243.548,-107.010,171.240,40.912,157.784
C05145=1040.987,243.797,-107.038,171.242,40.914,157.785
C05146=1040.994,244.045,-107.067,171.245,40.916,157.786
C05147=1041.000,244.294,-107.096,171.247,40.917,157.786
C05148=1041.007,244.541,-107.125,171.251,40.919,157.787
C05149=1041.013,244.790,-107.153,171.253,40.921,157.787
C05150=1041.020,245.039,-107.182,171.256,40.922,157.788
C05151=1041.027,245.287,-107.211,171.259,40.925,157.788
C05152=1041.033,245.535,-107.240,171.261,40.926,157.789
C05153=1041.039,245.783,-107.269,171.264,40.928,157.789
C05154=1041.045,246.031,-107.298,171.266,40.930,157.790
C05155=1041.052,246.279,-107.326,171.269,40.932,157.790
C05156=1041.059,246.528,-107.356,171.273,40.934,157.791
C05157=1041.065,246.776,-107.385,171.275,40.936,157.791
C05158=1041.072,247.024,-107.414,171.278,40.938,157.792
C05159=1041.078,247.272,-107.443,171.280,40.939,157.792
C05160=1041.084,247.520,-107.472,171.283,40.941,157.793
C05161=1041.091,247.769,-107.501,171.286,40.943,157.793
C05162=1041.098,248.017,-107.530,171.289,40.945,157.794
C05163=1041.104,248.265,-107.559,171.292,40.947,157.795
C05164=1041.112,248.565,-107.595,171.294,40.949,157.795
C05165=1041.120,248.864,-107.629,171.298,40.952,157.796
C05166=1041.128,249.163,-107.664,171.302,40.954,157.797
C05167=1041.136,249.462,-107.699,171.305,40.956,157.797
C05168=1041.143,249.711,-107.728,171.307,40.958,157.798
C05169=1041.149,249.959,-107.757,171.311,40.960,157.798
C05170=1041.155,250.207,-107.786,171.313,40.961,157.799
C05171=1041.161,250.455,-107.815,171.316,40.963,157.799
C05172=1041.168,250.704,-107.845,171.319,40.965,157.800
C05173=1041.175,250.951,-107.875,171.321,40.967,157.801
C05174=1041.182,251.199,-107.903,171.325,40.969,157.801
C05175=1041.189,251.448,-107.933,171.327,40.970,157.801
C05176=1041.195,251.696,-107.962,171.330,40.973,157.802
C05177=1041.201,251.944,-107.991,171.333,40.974,157.803
C05178=1041.208,252.193,-108.020,171.336,40.976,157.803
C05179=1041.214,252.441,-108.050,171.339,40.978,157.804
C05180=1041.221,252.689,-108.079,171.341,40.980,157.804
C05181=1041.228,252.938,-108.108,171.344,40.982,157.805
C05182=1041.234,253.186,-108.137,171.348,40.984,157.805
C05183=1041.241,253.433,-108.166,171.350,40.985,157.806
C05184=1041.248,253.682,-108.196,171.353,40.987,157.806
C05185=1041.254,253.930,-108.225,171.355,40.989,157.807
C05186=1041.261,254.179,-108.254,171.359,40.991,157.807
C05187=1041.268,254.426,-108.284,171.362,40.993,157.808
C05188=1041.274,254.674,-108.313,171.364,40.994,157.809
C05189=1041.281,254.923,-108.342,171.367,40.997,157.809
C05190=1041.287,255.171,-108.372,171.370,40.998,157.810
C05191=1041.294,255.420,-108.402,171.373,41.000,157.810
C05192=1041.300,255.668,-108.431,171.376,41.002,157.811
C05193=1041.307,255.916,-108.461,171.379,41.003,157.811
C05194=1041.314,256.164,-108.489,171.382,41.006,157.812
C05195=1041.321,256.411,-108.519,171.384,41.007,157.812
C05196=1041.328,256.660,-108.548,171.388,41.009,157.813
C05197=1041.334,256.908,-108.577,171.390,41.011,157.813
C05198=1041.341,257.156,-108.608,171.393,41.013,157.814
C05199=1041.348,257.405,-108.637,171.397,41.015,157.815
C05200=1041.355,257.653,-108.667,171.399,41.017,157.815
C05201=1041.361,257.901,-108.696,171.402,41.018,157.816
C05202=1041.368,258.149,-108.726,171.404,41.020,157.816
C05203=1041.374,258.397,-108.755,171.408,41.022,157.817
C05204=1041.382,258.646,-108.785,171.411,41.024,157.817
C05205=1041.388,258.894,-108.814,171.414,41.026,157.818
C05206=1041.395,259.142,-108.844,171.417,41.027,157.818
C05207=1041.402,259.390,-108.873,171.420,41.029,157.819
C05208=1041.409,259.638,-108.903,171.423,41.031,157.819
C05209=1041.416,259.887,-108.932,171.426,41.033,157.820
C05210=1041.422,260.134,-108.962,171.428,41.035,157.821
C05211=1041.429,260.383,-108.991,171.432,41.037,157.821
C05212=1041.436,260.631,-109.021,171.435,41.038,157.822
C05213=1041.443,260.879,-109.051,171.437,41.040,157.822
C05214=1041.449,261.127,-109.080,171.441,41.042,157.823
C05215=1041.456,261.375,-109.110,171.443,41.044,157.823
C05216=1041.463,261.624,-109.140,171.447,41.046,157.824
C05217=1041.470,261.871,-109.170,171.450,41.047,157.824
C05218=1041.477,262.120,-109.200,171.452,41.050,157.825
C05219=1041.484,262.367,-109.229,171.456,41.051,157.826
C05220=1041.491,262.665,-109.265,171.460,41.054,157.826
C05221=1041.499,262.963,-109.301,171.462,41.056,157.827
C05222=1041.507,263.261,-109.338,171.466,41.058,157.828
C05223=1041.515,263.559,-109.374,171.470,41.061,157.828
C05224=1041.521,263.807,-109.403,171.473,41.062,157.829
C05225=1041.529,264.055,-109.434,171.476,41.064,157.829
C05226=1041.535,264.303,-109.464,171.479,41.066,157.830
C05227=1041.541,264.551,-109.493,171.482,41.068,157.831
C05228=1041.548,264.800,-109.523,171.485,41.070,157.831
C05229=1041.554,265.047,-109.554,171.488,41.072,157.832
C05230=1041.561,265.296,-109.584,171.491,41.074,157.832
C05231=1041.569,265.544,-109.614,171.494,41.076,157.833
C05232=1041.574,265.792,-109.644,171.498,41.078,157.834
C05233=1041.582,266.040,-109.675,171.500,41.080,157.834
C05234=1041.588,266.287,-109.704,171.504,41.082,157.835
C05235=1041.595,266.536,-109.735,171.506,41.083,157.835
C05236=1041.602,266.784,-109.765,171.509,41.085,157.836
C05237=1041.608,267.032,-109.795,171.513,41.088,157.836
C05238=1041.615,267.280,-109.826,171.515,41.089,157.837
C05239=1041.622,267.528,-109.856,171.519,41.091,157.838
C05240=1041.628,267.776,-109.886,171.522,41.093,157.838
C05241=1041.635,268.024,-109.916,171.525,41.095,157.839
C05242=1041.642,268.273,-109.946,171.528,41.097,157.839
C05243=1041.648,268.521,-109.977,171.531,41.099,157.840
C05244=1041.655,268.769,-110.007,171.534,41.101,157.841
C05245=1041.662,269.017,-110.038,171.537,41.103,157.841
C05246=1041.668,269.264,-110.068,171.541,41.105,157.842
C05247=1041.675,269.513,-110.099,171.543,41.107,157.842
C05248=1041.682,269.761,-110.129,171.547,41.109,157.843
C05249=1041.688,270.009,-110.160,171.550,41.111,157.843
C05250=1041.695,270.257,-110.189,171.553,41.113,157.844
C05251=1041.701,270.505,-110.221,171.556,41.115,157.845
C05252=1041.709,270.753,-110.251,171.560,41.117,157.845
C05253=1041.714,271.001,-110.281,171.562,41.119,157.846
C05254=1041.722,271.249,-110.311,171.566,41.121,157.846
C05255=1041.728,271.497,-110.343,171.569,41.123,157.847
C05256=1041.735,271.745,-110.373,171.572,41.125,157.848
C05257=1041.741,271.993,-110.403,171.575,41.127,157.848
C05258=1041.748,272.241,-110.435,171.579,41.129,157.849
C05259=1041.755,272.489,-110.465,171.581,41.131,157.849
C05260=1041.762,272.738,-110.496,171.585,41.133,157.850
C05261=1041.768,272.985,-110.527,171.588,41.135,157.851
C05262=1041.775,273.233,-110.557,171.591,41.136,157.851
C05263=1041.781,273.482,-110.587,171.594,41.139,157.852
C05264=1041.788,273.729,-110.619,171.598,41.141,157.853
C05265=1041.795,273.977,-110.649,171.600,41.143,157.853
C05266=1041.801,274.225,-110.680,171.604,41.145,157.854
C05267=1041.808,274.473,-110.711,171.607,41.147,157.854
C05268=1041.815,274.721,-110.742,171.610,41.149,157.855
C05269=1041.822,274.970,-110.772,171.613,41.151,157.856
C05270=1041.828,275.217,-110.804,171.617,41.153,157.856
C05271=1041.835,275.465,-110.834,171.619,41.155,157.857
C05272=1041.842,275.713,-110.865,171.623,41.157,157.857
C05273=1041.848,275.961,-110.896,171.626,41.159,157.858
C05274=1041.855,276.209,-110.927,171.630,41.161,157.859
C05275=1041.862,276.457,-110.957,171.632,41.163,157.859
C05276=1041.870,276.760,-110.995,171.637,41.165,157.860
C05277=1041.878,277.061,-111.033,171.641,41.168,157.861
C05278=1041.886,277.364,-111.071,171.645,41.171,157.862
C05279=1041.894,277.666,-111.109,171.649,41.173,157.862
C05280=1041.900,277.915,-111.140,171.651,41.175,157.863
C05281=1041.908,278.162,-111.170,171.655,41.177,157.864
C05282=1041.915,278.410,-111.202,171.659,41.179,157.864
C05283=1041.921,278.659,-111.233,171.661,41.181,157.865
C05284=1041.928,278.906,-111.264,171.665,41.183,157.865
C05285=1041.934,279.154,-111.295,171.668,41.185,157.866
C05286=1041.941,279.402,-111.326,171.671,41.188,157.867
C05287=1041.947,279.650,-111.357,171.675,41.190,157.867
C05288=1041.954,279.898,-111.389,171.678,41.192,157.868
C05289=1041.960,280.146,-111.420,171.682,41.194,157.869
C05290=1041.967,280.394,-111.451,171.684,41.196,157.869
C05291=1041.974,280.642,-111.483,171.688,41.198,157.870
C05292=1041.981,280.890,-111.514,171.691,41.200,157.871
C05293=1041.987,281.138,-111.545,171.694,41.202,157.871
C05294=1041.994,281.386,-111.576,171.698,41.204,157.872
C05295=1042.001,281.634,-111.608,171.701,41.206,157.872
C05296=1042.007,281.882,-111.639,171.705,41.208,157.873
C05297=1042.014,282.130,-111.671,171.708,41.211,157.874
C05298=1042.021,282.378,-111.702,171.711,41.213,157.874
C05299=1042.027,282.626,-111.734,171.715,41.215,157.875
C05300=1042.034,282.873,-111.765,171.717,41.217,157.876
C05301=1042.041,283.121,-111.796,171.721,41.219,157.876
C05302=1042.048,283.369,-111.828,171.725,41.221,157.877
C05303=1042.054,283.617,-111.859,171.728,41.223,157.878
C05304=1042.061,283.865,-111.891,171.732,41.226,157.878
C05305=1042.068,284.113,-111.922,171.735,41.228,157.879
C05306=1042.075,284.361,-111.954,171.738,41.230,157.880
C05307=1042.081,284.609,-111.985,171.742,41.232,157.880
C05308=1042.088,284.857,-112.017,171.745,41.234,157.881
C05309=1042.095,285.105,-112.048,171.748,41.236,157.882
C05310=1042.101,285.352,-112.079,171.752,41.238,157.882
C05311=1042.108,285.600,-112.112,171.756,41.240,157.883
C05312=1042.115,285.848,-112.143,171.758,41.243,157.884
C05313=1042.122,286.096,-112.174,171.762,41.245,157.884
C05314=1042.129,286.343,-112.206,171.766,41.247,157.885
C05315=1042.135,286.591,-112.237,171.769,41.249,157.886
C05316=1042.142,286.839,-112.269,171.772,41.251,157.886
C05317=1042.149,287.087,-112.301,171.776,41.253,157.887
C05318=1042.156,287.334,-112.332,171.780,41.255,157.888
C05319=1042.162,287.583,-112.365,171.782,41.258,157.888
C05320=1042.169,287.831,-112.396,171.786,41.260,157.889
C05321=1042.176,288.079,-112.428,171.790,41.262,157.890
C05322=1042.183,288.326,-112.460,171.793,41.264,157.890
C05323=1042.189,288.575,-112.492,171.797,41.267,157.891
C05324=1042.196,288.822,-112.524,171.800,41.269,157.892
C05325=1042.203,289.070,-112.555,171.804,41.271,157.892
C05326=1042.209,289.318,-112.587,171.807,41.273,157.893
C05327=1042.217,289.566,-112.619,171.811,41.275,157.894
C05328=1042.223,289.814,-112.651,171.814,41.277,157.894
C05329=1042.230,290.061,-112.683,171.818,41.279,157.895
C05330=1042.237,290.309,-112.715,171.821,41.282,157.896
C05331=1042.243,290.557,-112.748,171.825,41.284,157.896
C05332=1042.252,290.871,-112.788,171.830,41.287,157.897
C05333=1042.260,291.185,-112.829,171.834,41.290,157.898
C05334=1042.269,291.500,-112.869,171.839,41.292,157.899
C05335=1042.277,291.813,-112.910,171.842,41.295,157.900
C05336=1042.285,292.061,-112.942,171.846,41.298,157.901
C05337=1042.291,292.309,-112.974,171.850,41.300,157.901
C05338=1042.298,292.557,-113.006,171.853,41.302,157.902
C05339=1042.304,292.805,-113.038,171.857,41.305,157.903
C05340=1042.311,293.052,-113.070,171.860,41.307,157.903
C05341=1042.318,293.300,-113.103,171.864,41.309,157.904
C05342=1042.325,293.548,-113.134,171.867,41.311,157.905
C05343=1042.331,293.796,-113.167,171.871,41.313,157.905
C05344=1042.338,294.043,-113.199,171.875,41.315,157.906
C05345=1042.346,294.291,-113.231,171.878,41.318,157.907
C05346=1042.352,294.539,-113.264,171.882,41.320,157.908
C05347=1042.359,294.786,-113.296,171.885,41.323,157.908
C05348=1042.366,295.035,-113.328,171.889,41.325,157.909
C05349=1042.373,295.283,-113.361,171.893,41.327,157.910
C05350=1042.379,295.530,-113.393,171.896,41.330,157.910
C05351=1042.386,295.777,-113.425,171.900,41.332,157.911
C05352=1042.393,296.026,-113.459,171.904,41.334,157.912
C05353=1042.399,296.273,-113.491,171.907,41.336,157.913
C05354=1042.405,296.521,-113.524,171.911,41.339,157.913
C05355=1042.412,296.768,-113.557,171.915,41.342,157.914
C05356=1042.419,297.016,-113.589,171.918,41.344,157.915
C05357=1042.426,297.264,-113.622,171.922,41.346,157.916
C05358=1042.432,297.512,-113.654,171.925,41.348,157.916
C05359=1042.438,297.760,-113.687,171.929,41.351,157.917
C05360=1042.446,298.007,-113.720,171.933,41.353,157.918
C05361=1042.452,298.255,-113.753,171.937,41.356,157.919
C05362=1042.458,298.502,-113.786,171.940,41.358,157.919
C05363=1042.465,298.751,-113.819,171.944,41.360,157.920
C05364=1042.472,298.998,-113.851,171.947,41.363,157.921
C05365=1042.479,299.246,-113.884,171.951,41.365,157.921
C05366=1042.486,299.494,-113.917,171.955,41.368,157.922
C05367=1042.492,299.741,-113.949,171.959,41.370,157.923
C05368=1042.498,299.989,-113.982,171.962,41.372,157.924
C05369=1042.505,300.237,-114.015,171.966,41.375,157.924
C05370=1042.512,300.485,-114.047,171.970,41.377,157.925
C05371=1042.519,300.732,-114.081,171.973,41.380,157.926
C05372=1042.526,300.980,-114.114,171.977,41.382,157.927
C05373=1042.532,301.227,-114.147,171.981,41.385,157.928
C05374=1042.539,301.476,-114.180,171.984,41.387,157.928
C05375=1042.546,301.723,-114.212,171.988,41.389,157.929
C05376=1042.553,301.971,-114.246,171.992,41.392,157.930
C05377=1042.559,302.218,-114.279,171.996,41.394,157.930
C05378=1042.566,302.466,-114.311,172.000,41.397,157.931
C05379=1042.573,302.714,-114.345,172.004,41.399,157.932
C05380=1042.580,302.961,-114.377,172.008,41.401,157.933
C05381=1042.587,303.209,-114.410,172.012,41.404,157.934
C05382=1042.593,303.456,-114.444,172.014,41.407,157.934
C05383=1042.600,303.704,-114.477,172.018,41.409,157.935
C05384=1042.606,303.952,-114.510,172.022,41.411,157.936
C05385=1042.614,304.200,-114.543,172.026,41.414,157.937
C05386=1042.621,304.447,-114.576,172.030,41.417,157.937
C05387=1042.628,304.695,-114.609,172.034,41.419,157.938
C05388=1042.637,305.026,-114.653,172.039,41.422,157.939
C05389=1042.646,305.356,-114.698,172.044,41.425,157.940
C05390=1042.655,305.687,-114.742,172.049,41.428,157.941
C05391=1042.664,306.017,-114.787,172.054,41.432,157.942
C05392=1042.671,306.265,-114.820,172.058,41.435,157.943
C05393=1042.678,306.512,-114.853,172.062,41.437,157.944
C05394=1042.685,306.760,-114.886,172.066,41.439,157.945
C05395=1042.692,307.007,-114.919,172.070,41.442,157.945
C05396=1042.699,307.255,-114.953,172.074,41.444,157.946
C05397=1042.706,307.503,-114.986,172.078,41.447,157.947
C05398=1042.713,307.750,-115.019,172.082,41.449,157.948
C05399=1042.720,307.999,-115.053,172.085,41.452,157.948
C05400=1042.726,308.246,-115.086,172.089,41.454,157.949
C05401=1042.734,308.493,-115.119,172.093,41.457,157.950
C05402=1042.741,308.741,-115.152,172.097,41.459,157.951
C05403=1042.748,308.989,-115.186,172.101,41.462,157.952
C05404=1042.755,309.236,-115.220,172.105,41.464,157.952
